(* IEC 61131-3 sources: elnaProjects/kc6/build_BaseProject_ecl/_ (part 5) *)

  (* [A2-14, AI0-1] T_medi_statora_faza_2 *)
  stAI_Ini(data_Ini := TRUE,  dLL := 0.0, dHL := 150.0,
  ISVALIDREF_HW := TRUE, dHW := 130.0, aperturFilter:= 0.5,
  strAI := ai.TStalisStatoraKanal2);
  inits := inits + BOOL_TO_UINT(stAI_Ini.Init);

  (* [A2-14, AI0-2] T_medi_statora_faza_3 *)
  stAI_Ini(data_Ini := TRUE,  dLL := 0.0, dHL :=150.0,
  ISVALIDREF_HW := TRUE, dHW := 130.0, aperturFilter:= 0.5,
  strAI := ai.TStalisStatoraKanal3);
  inits := inits + BOOL_TO_UINT(stAI_Ini.Init);

  (* [A2-14, AI0-3] T_stali_statora_faza_1 *)
  stAI_Ini(data_Ini := TRUE,  dLL := 0.0, dHL := 150.0,
  ISVALIDREF_HW := TRUE, dHW := 130.0, aperturFilter:= 0.5,
  strAI := ai.TMediStatoraKanal1);
  inits := inits + BOOL_TO_UINT(stAI_Ini.Init);

  (********************************************* Модуль A2-15 ******************************************************)

  (* [A2-15, AI1-0] T_stali_statora_faza_2 *)
  stAI_Ini(data_Ini :=TRUE,  dLL := 0.0, dHL := 150.0,
  ISVALIDREF_HW := TRUE, dHW := 130.0, aperturFilter:= 0.5,
  strAI := ai.TMediStatoraKanal2);
  inits := inits + BOOL_TO_UINT(stAI_Ini.Init);

  (* [A2-15, AI1-1] T_stali_statora_faza_3 *)
  stAI_Ini(data_Ini := TRUE,  dLL := 0.0, dHL := 150.0,
  ISVALIDREF_HW := TRUE, dHW := 130.0, aperturFilter:= 0.5,
  strAI := ai.TMediStatoraKanal3);
  inits := inits + BOOL_TO_UINT(stAI_Ini.Init);

  (* [A2-15, AI1-2] T_goryachego_vozdyha_ed_t1 *)
  stAI_Ini(data_Ini := TRUE,  dLL := 0.0, dHL := 100.0,
  ISVALIDREF_HW := TRUE, dHW := 70.0, aperturFilter:= 0.5,
  strAI := ai.TOpornogoPodshipnikaEDT_1);
  inits := inits + BOOL_TO_UINT(stAI_Ini.Init);

  (* [A2-15, AI1-3]  T_goryachego_vozdyha_ed_t2 *)
  stAI_Ini(data_Ini := TRUE,  dLL := 0.0, dHL := 100.0,
  ISVALIDREF_HW := TRUE, dHW := 70.0, aperturFilter:= 0.5,
  strAI := ai.TOpornoYpornogoPodshipnikaEDT_2);
  inits := inits + BOOL_TO_UINT(stAI_Ini.Init);

  (********************************************* Модуль A3-1 ******************************************************)

  (* [A3-1, AI2-0]  T_holodnogo_vozdyha_ed_t1 *)
  stAI_Ini(data_Ini := TRUE,  dLL := 0.0, dHL := 100.0,
  ISVALIDREF_HW := TRUE, dHW := 70.0, aperturFilter:= 0.5,
  strAI := ai.TOpornoYpornogoPodshipnikaKolesaRedEDT_3);
  inits := inits + BOOL_TO_UINT(stAI_Ini.Init);

  (* [A3-1, AI2-1] T_holodnogo_vozdyha_ed_t2 *)
  stAI_Ini(data_Ini := TRUE,  dLL := 0.0, dHL := 100.0,
  ISVALIDREF_HW := TRUE, dHW := 70.0, aperturFilter:= 0.5,
  strAI := ai.TOpornoYpornogoPodshipnikaKolesaRedHT_4);
  inits := inits + BOOL_TO_UINT(stAI_Ini.Init);

  (* [A3-1, AI2-2] T_opornogo_podshipnika_electro_dvigatelia_t1 *)
  stAI_Ini(data_Ini := TRUE,  dLL := 0.0, dHL := 100.0,
  ISVALIDREF_HA := TRUE, ISVALIDREF_HW := TRUE, dHA := 80.0, dHW := 75.0, aperturFilter:= 0.5,
  strAI := ai.TOpornogoPodshipnikaShesterniReduktoraT_5);
  inits := inits + BOOL_TO_UINT(stAI_Ini.Init);

  (* [A3-1, AI2-3] T_opornogo_ypornogo_podshipnika_electro_dvigatelia_so_storony_redyctora_t2 *)
  stAI_Ini(data_Ini := TRUE,  dLL := 0.0, dHL := 100.0,
  ISVALIDREF_HA := TRUE, ISVALIDREF_HW := TRUE, dHA := 80.0, dHW := 75.0, aperturFilter:= 0.5,
  strAI := ai.TOpornogoPodshipnikaReduktoraHT_6);
  inits := inits + BOOL_TO_UINT(stAI_Ini.Init);

  (********************************************* Модуль A3-2 ******************************************************)

  (* [A3-2, AI3-01]  T_oporno_ypornogo_podshipnika_kolesa_redyctora_so_storony_electro_dvigatelya_t3 *)
  stAI_Ini(data_Ini := TRUE,  dLL := 0.0, dHL := 100.0,
  ISVALIDREF_HA := TRUE, ISVALIDREF_HW := TRUE, dHA := 80.0, dHW := 75.0, aperturFilter:= 0.5,
  strAI := ai.TOpornoYpornogoPodshipnikaNagnetateljaT_7_1);
  inits := inits + BOOL_TO_UINT(stAI_Ini.Init);

  (* [A3-2, AI3-1]  T_opornogo_podshipnika_kolesa_redyctora_so_storony_nagnetatelya_t4 *)
  stAI_Ini(data_Ini := TRUE,  dLL := 0.0, dHL := 100.0, aperturFilter:= 0.5,
  ISVALIDREF_HA := TRUE, ISVALIDREF_HW := TRUE, dHA := 80.0, dHW := 75.0,
  strAI := ai.TOpornoYpornogoPodshipnikaNagnetateljaT_7_2);
  inits := inits + BOOL_TO_UINT(stAI_Ini.Init);

  (* [A3-2, AI3-2]  Т подшипника редуктора, т4 *)
  stAI_Ini(data_Ini := TRUE,  dLL := 0.0, dHL := 100.0,
  ISVALIDREF_HA := TRUE, ISVALIDREF_HW := TRUE, dHA := 80.0, dHW := 75.0, aperturFilter:= 0.5,
  strAI := ai.TOpornoYpornogoPodshipnikaSvobodnogoKoncaNT_8_1);
  inits := inits + BOOL_TO_UINT(stAI_Ini.Init);

  (* [A3-2, AI3-3]  Т опорного подшипника нагнетателя, т1 *)
  stAI_Ini(data_Ini := TRUE,  dLL := 0.0, dHL := 100.0,
  ISVALIDREF_HA := TRUE, ISVALIDREF_HW := TRUE, dHA := 80.0, dHW := 75.0, aperturFilter:= 0.5,
  strAI := ai.TOpornoYpornogoPodshipnikaSvobodnogoKoncaNT_8_2);
  inits := inits + BOOL_TO_UINT(stAI_Ini.Init);

  (********************************************* Модуль A3-3 ******************************************************)

  (* [A3-3, AI4-1]  T_oporno_ypornogo_podshipnika_nagnetatelya_so_storony_redyctora_t7_osnovnoi *)
  stAI_Ini(data_Ini := TRUE,  dLL := 0.0, dHL := 100.0,
  ISVALIDREF_HA := TRUE, ISVALIDREF_HW := TRUE, dHA := 80.0, dHW := 75.0, aperturFilter:= 0.5,
  strAI := ai.TYpornogoPodshipnikaRavKolodokHT_9_1);
  inits := inits + BOOL_TO_UINT(stAI_Ini.Init);

  (* [A3-3, AI4-2]  T_oporno_ypornogo_podshipnika_nagnetatelya_so_storony_redyctora_t7_rezervniy *)
  stAI_Ini(data_Ini := TRUE,  dLL := 0.0, dHL := 100.0,
  ISVALIDREF_HA := TRUE, ISVALIDREF_HW := TRUE, dHA := 80.0, dHW := 75.0, aperturFilter:= 0.5,
  strAI := ai.TYpornogoPodshipnikaRavKolodokHT_9_2);
  inits := inits + BOOL_TO_UINT(stAI_Ini.Init);

  (* [A3-3, AI4-3] T_oporno_ypornogo_podshipnika_svobodnogo_konca_nagnetatelya_t8_osnovnoi *)
  stAI_Ini(data_Ini := TRUE,  dLL := 0.0, dHL := 100.0,
  ISVALIDREF_HA := TRUE, ISVALIDREF_HW := TRUE, dHA := 80.0, dHW := 75.0, aperturFilter:= 0.5,
  strAI := ai.TYpornogoPodshipnikaNerabKolodokHT_10_1);
  inits := inits + BOOL_TO_UINT(stAI_Ini.Init);

  (* [A3-3, AI4-4] T_oporno_ypornogo_podshipnika_svobodnogo_konca_nagnetatelya_t8_rezervniy *)
  stAI_Ini(data_Ini := TRUE,  dLL := 0.0, dHL := 100.0,
  ISVALIDREF_HA := TRUE, ISVALIDREF_HW := TRUE, dHA := 80.0, dHW := 75.0, aperturFilter:= 0.5,
  strAI := ai.TYpornogoPodshipnikaNerabKolodokHT_10_2);
  inits := inits + BOOL_TO_UINT(stAI_Ini.Init);

  (********************************************* Модуль A3-4 ******************************************************)

  (* [A3-4, AI5-0] T_ypornogo_podshipnika_rabochih_kolodok_nagnetatelya_t9 *)
  stAI_Ini(data_Ini := TRUE,  dLL := 0.0, dHL := 100.0,
  ISVALIDREF_HA := TRUE, ISVALIDREF_HW := TRUE, dHA := 80.0, dHW := 75.0, aperturFilter:= 0.5,
  strAI := ai.THolodnogoVozduhaEDKanall);
  inits := inits + BOOL_TO_UINT(stAI_Ini.Init);

  (* [A3-4, AI5-1] T_ne_rabochih_kolodok_ypornogo_podshipnika_nagnetatelya_t10 *)
  stAI_Ini(data_Ini := TRUE,  dLL := 0.0, dHL := 100.0,
  ISVALIDREF_HA := TRUE, ISVALIDREF_HW := TRUE, dHA := 80.0, dHW := 75.0, aperturFilter:= 0.5,
  strAI := ai.THolodnogoVozduhaEDKanal2);
  inits := inits + BOOL_TO_UINT(stAI_Ini.Init);

  (* [A3-4, AI5-2]  T_gaz_in_nagnetatelia *)
  stAI_Ini(data_Ini := TRUE,  dLL := -50.0, dHL := 100.0,
  ISVALIDREF_HW := TRUE, dHW := 80.0, aperturFilter:= 0.5,
  strAI := ai.TGorjachegoVozduhaEDKanall);
  inits := inits + BOOL_TO_UINT(stAI_Ini.Init);

  (* [A3-4, AI5-3] T_gaz_out_nagnetatelia *)
  stAI_Ini(data_Ini := TRUE,  dLL := -50.0, dHL := 100.0,
  ISVALIDREF_HA := TRUE, ISVALIDREF_HW := TRUE, dHA := 90.0, dHW := 80.0, aperturFilter:= 0.5,
  strAI := ai.TGorjachegoVozduhaEDKanal2);
  inits := inits + BOOL_TO_UINT(stAI_Ini.Init);

  (********************************************* Модуль A3-5 ******************************************************)

  (* [A3-5, AI6-0] T_masla_do_ABO *)
  stAI_Ini(data_Ini := TRUE,  dLL := 0.0, dHL := 100.0,
  ISVALIDREF_HW := TRUE, dHW := 55.0, aperturFilter:= 0.5,
  strAI := ai.TNArujnogoVozduha);
  inits := inits + BOOL_TO_UINT(stAI_Ini.Init);

  (* [A3-5, AI6-1]  T_masla_posle_ABO *)
  stAI_Ini(data_Ini := TRUE,  dLL := 0.0, dHL := 100.0,
  ISVALIDREF_HW := TRUE, dHW := 55.0, aperturFilter:= 0.5,
  strAI := ai.TgazaNaVhodeH);
  inits := inits + BOOL_TO_UINT(stAI_Ini.Init);

  (* [A3-5, AI6-2] T_masla_v_maslobake *)
  stAI_Ini(data_Ini := TRUE,  dLL := 0.0, dHL := 100.0,
  ISVALIDREF_LW := TRUE, dLW := 25.0, aperturFilter:= 0.5,
  strAI := ai.TgazaNaVyhodeH);
  inits := inits + BOOL_TO_UINT(stAI_Ini.Init);

  (********************************************* Модуль A3-6 ******************************************************)

  (* [A3-6, AI7-0] T_masla_v_maslobake_nad_ten *)
  stAI_Ini(data_Ini := TRUE,  dLL := 0.0, dHL := 100.0,
  ISVALIDREF_HW := TRUE, dHW := 60.0, aperturFilter:= 0.5,
  strAI := ai.T_masla_v_maslobake_nad_ten);
  inits := inits + BOOL_TO_UINT(stAI_Ini.Init);

  (* [A3-6, AI7-1] T_naryjnogo_vozdyxa_rezervniy *)
  stAI_Ini(data_Ini := TRUE,  dLL := -50.0, dHL := 100.0,
  aperturFilter:= 0.5,
  strAI := ai.T_naryjnogo_vozdyxa);
  inits := inits + BOOL_TO_UINT(stAI_Ini.Init);

  (* [A3-6, AI7-2] T_vozduha_V_shkafy *)
  stAI_Ini(data_Ini := TRUE,  dLL := -50.0, dHL := 100.0,
  aperturFilter:= 0.5,
  strAI := ai.T_vozduha_V_shkaf);
  inits := inits + BOOL_TO_UINT(stAI_Ini.Init);

  (********************************************* Модуль A3-8 ******************************************************)

  (* [A3-8, AI9-0]  Davlenie_impylsnogo_gaza *)
  stAI_Ini(data_Ini := TRUE,  dLL := 0.0, dHL := 10.0,
  ISVALIDREF_LW := TRUE, dLW := 5.0, aperturFilter:= 0.5,
  strAI := ai.Davlenie_impylsnogo_gaza);
  inits := inits + BOOL_TO_UINT(stAI_Ini.Init);

  (* [A3-8, AI9-1]  Yroven_masla_v_maslobake *)
  stAI_Ini(data_Ini := TRUE,  dLL := 340.0, dHL := 960.0,
  ISVALIDREF_LW := TRUE, dLW := 350.0, aperturFilter:= 0.5,
  strAI := ai.Yroven_masla_v_maslobake);
  inits := inits + BOOL_TO_UINT(stAI_Ini.Init);

  (* [A3-8, AI9-2]  Osevoi_sdvig_nagnetatelya_vpravo *)
  stAI_Ini(data_Ini := TRUE,  dLL := 0.0, dHL := 1000.0,
  ISVALIDREF_HA := TRUE, ISVALIDREF_HW := TRUE, dHA := 300.0, dHW := 200.0, aperturFilter:= 0.5,
  strAI := ai.Osevoi_sdvig_nagnetatelya_vpravo);
  inits := inits + BOOL_TO_UINT(stAI_Ini.Init);

  (* [A3-8, AI9-3]  Osevoi_sdvig_nagnetatelya_vlevo *)
  stAI_Ini(data_Ini := TRUE,  dLL := 0.0, dHL := 1000.0,
  ISVALIDREF_LA := TRUE, ISVALIDREF_LW := TRUE, dHA := 300.0, dHW := 200.0, aperturFilter:= 0.5,
  strAI := ai.Osevoi_sdvig_nagnetatelya_vlevo);
  inits := inits + BOOL_TO_UINT(stAI_Ini.Init);

  (********************************************* Модуль A3-9 ******************************************************)

  (* [A3-9, AI10-0]  Tok_statora *)
  stAI_Ini(data_Ini := TRUE,  dLL := 0.0, dHL := 1000.0,
  ISVALIDREF_LW := TRUE, dLW := 240.0, aperturFilter:= 0.5,
  strAI := ai.Tok_statora);
  inits := inits + BOOL_TO_UINT(stAI_Ini.Init);

  (* [A3-9, AI10-1]  Kontrol_220_perem *)
  stAI_Ini(data_Ini := TRUE,  dLL := 0.0, dHL := 250.0, aperturFilter:= 0.5,
  ISVALIDREF_LW := TRUE, ISVALIDREF_HW := TRUE,
  dLW := 187.0, dHW := 242.0,
  strAI := ai.Kontrol_220_perem);
  inits := inits + BOOL_TO_UINT(stAI_Ini.Init);

  (* [A3-9, AI10-2] Kontrol_220_post *)
  stAI_Ini(data_Ini := TRUE,  dLL := 0.0, dHL := 250.0, aperturFilter:= 0.5,
  ISVALIDREF_LW := TRUE, ISVALIDREF_HW := TRUE,
  dLW := 187.0, dHW := 242.0,
  strAI := ai.Kontrol_220_post);
  inits := inits + BOOL_TO_UINT(stAI_Ini.Init);

  (********************************************* Модуль A3-10 ******************************************************)

  (* [A3-10, AI11-0] Davlenie_gaza_na_vhode_nagnetatelya *)
  stAI_Ini(data_Ini := TRUE,  dLL := 0.0, dHL := 10.0,
  ISVALIDREF_LW := TRUE, dLW := 5.0, (*ISVALIDREF_LA := TRUE, dLA := 4.6,*) aperturFilter:= 0.5,
  strAI := ai.Davlenie_gaza_na_vhode_nagnetatelya);
  inits := inits + BOOL_TO_UINT(stAI_Ini.Init);

  (* [A3-10, AI11-1] Davlenie_gaza_na_vihode_nagnetatelya *)
  stAI_Ini(data_Ini := TRUE,  dLL := 0.0, dHL := 10.0,
  ISVALIDREF_HW := TRUE, dHW := 7.55, (*ISVALIDREF_HA := TRUE, dHA := 7.65,*) aperturFilter:= 0.5,
  strAI := ai.Davlenie_gaza_na_vihode_nagnetatelya);
  inits := inits + BOOL_TO_UINT(stAI_Ini.Init);

  (* [A3-10, AI11-2] Perepad_davleniya_maslo_gaz *)
  stAI_Ini(data_Ini := TRUE,  dLL := 0.0, dHL := 1600.0,
  ISVALIDREF_LW := TRUE, dLW := 150.0, ISVALIDREF_LA := TRUE, dLA := 100.0,
  strAI := ai.Perepad_davleniya_maslo_gaz);
  inits := inits + BOOL_TO_UINT(stAI_Ini.Init);

  (* [A3-10, AI11-3] Davlenie_masla_posle_nasosa_yplotneniya *)
  stAI_Ini(data_Ini := TRUE,  dLL := 0.0, dHL := 10.0, aperturFilter:= 0.5,
  strAI := ai.Davlenie_masla_posle_nasosa_yplotneniya);
  inits := inits + BOOL_TO_UINT(stAI_Ini.Init);

  (********************************************* Модуль A3-11 ******************************************************)

  (* [A3-11, AI12-0]  Davlenie_masla_smazki_nizkoe *)
  stAI_Ini(data_Ini := TRUE,  dLL := 0.0, dHL := 1000.0,
  ISVALIDREF_LW := TRUE, dLW := 50.0, ISVALIDREF_LA := TRUE, dLA := 25.0,
  strAI := ai.Davlenie_masla_smazki_nizkoe);
  inits := inits + BOOL_TO_UINT(stAI_Ini.Init);

  (* [A3-11, AI12-1]  Davlenie_masla_smazki_visokoe *)
  stAI_Ini(data_Ini := TRUE,  dLL := 0.0, dHL := 1000.0,
  ISVALIDREF_LW := TRUE, dLW := 300.0, ISVALIDREF_LA := TRUE, dLA := 250.0,
  strAI := ai.Davlenie_masla_smazki_visokoe);
  inits := inits + BOOL_TO_UINT(stAI_Ini.Init);

  (* [A3-11, AI12-2]  Davlenie_masla_smazki_posle_GNS *)
  stAI_Ini(data_Ini := TRUE,  dLL := 0.0, dHL := 1000.0,
  ISVALIDREF_LW := TRUE, dLW := 400.0, aperturFilter:= 0.5,
  strAI := ai.Davlenie_masla_smazki_posle_GNS);
  inits := inits + BOOL_TO_UINT(stAI_Ini.Init);

  (* [A3-11, AI12-3]  Perepad_davleniya_gaza_na_konfyzore *)
  stAI_Ini(data_Ini := TRUE,  dLL := 0.0, dHL := 250.0, aperturFilter:= 0.5,
  strAI := ai.Perepad_davleniya_gaza_na_konfyzore);
  inits := inits + BOOL_TO_UINT(stAI_Ini.Init);

  (********************************************* Модуль A3-12 ******************************************************)

  (* [A3-12, AI13-0] Perepad_davleniya_masla_na_maslyanom_filtre *)
  stAI_Ini(data_Ini := TRUE,  dLL := 0.0, dHL := 250.0,
  ISVALIDREF_HW := TRUE, dHW := 150.0, aperturFilter:= 0.5,
  strAI := ai.Perepad_davleniya_masla_na_maslyanom_filtre);
  inits := inits + BOOL_TO_UINT(stAI_Ini.Init);

  (********************************************* Модуль A3-13 ******************************************************)

  (* [A3-13, AI14-0]  Vibroploskost_opornogo_podshipnika_electro_dvigatelya_t1 *)
  stAI_Ini(data_Ini := TRUE,  dLL := 0.0, dHL := 25.0,
  ISVALIDREF_HW := TRUE, ISVALIDREF_HA := TRUE, dHW := 11.0, dHA := 18.0,
  strAI := ai.Vibroskorost_OP_ED_t1);
  inits := inits + BOOL_TO_UINT(stAI_Ini.Init);

  (* [A3-13, AI14-1]  Vibroploskost_oporno_ypornogo_podshipnika_electro_dvigatelya_so_storony_redyctora_t2 *)
  stAI_Ini(data_Ini := TRUE,  dLL := 0.0, dHL := 25.0,
  ISVALIDREF_HW := TRUE, ISVALIDREF_HA := TRUE, dHW := 11.0, dHA := 18.0, aperturFilter:= 0.5,
  strAI := ai.Vibroskorost_OYP_ED_so_storony_redyctora_t2);
  inits := inits + BOOL_TO_UINT(stAI_Ini.Init);

  (* [A3-13, AI14-2]  Vibroploskost_oporno_ypornogo_podshipnika_kolesa_redyktora_so_storony_electro_dvigatelya_t3 *)
  stAI_Ini(data_Ini := TRUE,  dLL := 0.0, dHL := 25.0,
  ISVALIDREF_HW := TRUE, ISVALIDREF_HA := TRUE, dHW := 11.0, dHA := 18.0, aperturFilter:= 0.5,
  strAI := ai.Vibroskorost_OYP_kolesa_ED_t3);
  inits := inits + BOOL_TO_UINT(stAI_Ini.Init);

  (* [A3-13, AI14-3]  Vibroploskost_oporno_ypornogo_podshipnika_kolesa_redyktora_so_storony_nagnetatelya_t4_rezerv *)
  stAI_Ini(data_Ini := TRUE,  dLL := 0.0, dHL := 25.0,
  ISVALIDREF_HW := TRUE, ISVALIDREF_HA := TRUE, dHW := 11.0, dHA := 18.0, aperturFilter:= 0.5,
  strAI := ai.Vibroskorost_OP_kolesa_nagnetatelya_t4);
  inits := inits + BOOL_TO_UINT(stAI_Ini.Init);

  (********************************************* Модуль A3-14 ******************************************************)

  (* [A3-14, AI15-0]  Vibroploskost_opornogo_podshipnika_shesterni_redyktora_so_storony_nagnetatelya_t5_rezerv *)
  stAI_Ini(data_Ini := TRUE,  dLL := 0.0, dHL := 25.0,
  ISVALIDREF_HW := TRUE, ISVALIDREF_HA := TRUE, dHW := 11.0, dHA := 18.0, aperturFilter:= 0.5,
  strAI := ai.Vibroskorost_OP_shesterni_ED_t5);
  inits := inits + BOOL_TO_UINT(stAI_Ini.Init);

  (* [A3-14, AI15-1]  Vibroploskost_opornogo_podshipnika_shesterni_redyktora_so_storony_nagnetatelya_t6 *)
  stAI_Ini(data_Ini := TRUE,  dLL := 0.0, dHL := 25.0,
  ISVALIDREF_HW := TRUE, ISVALIDREF_HA := TRUE, dHW := 11.0, dHA := 18.0, aperturFilter:= 0.5,
  strAI := ai.Vibroskorost_OP_shesterni_nagnetatelya_t6);
  inits := inits + BOOL_TO_UINT(stAI_Ini.Init);

  initiales := 0;
  IF init THEN initiales := inits; END_IF;
END_FUNCTION_BLOCK

FUNCTION_BLOCK proc_AO
  VAR
    fb_Reserv_AO_1 : fb_AOSourceMlp;
    fb_Reserv_AO_2 : fb_AOSourceMlp;
  END_VAR
  VAR_EXTERNAL
    ao : AOConfig;
    arAOUT_0 : TDoubleData;
    arAOUT_1 : TDoubleData;
  END_VAR

  (* Циклический опрос. Входные аналоговые параметры *)

  (* Модуль A10 *)

  (* [A10-1, AO0] Резерв (A10) *)
  fb_Reserv_AO_1(OutCurrent := arAOUT_0, strAO := ao.Reserv_AO_1);

  (* [A10-1, AO1] Резерв (A10) *)
  fb_Reserv_AO_2(OutCurrent := arAOUT_1, strAO := ao.Reserv_AO_2);
END_FUNCTION_BLOCK

FUNCTION_BLOCK proc_AO_Init
  VAR_INPUT
    init : BOOL;
  END_VAR
  VAR
    stAO_Ini : fb_AO_Init;
    inits : UINT;
  END_VAR
  VAR_INPUT
    initiales : UINT;
  END_VAR
  VAR_EXTERNAL
    ao : AOConfig;
  END_VAR

  (* Инициализация начало. Входные аналоговые параметры *)

  inits := 0; (* Флаг необходимости инициализации структур-дескрипторов *)

  (* Модуль A10 *)
  (* [A10, AO0] Резерв (A) *)
  stAO_Ini(data_Ini := TRUE, (*outLL := 4000.0, outHL := 20000.0,*)
    newLL_ISVALIDREF := TRUE, newHL_ISVALIDREF := TRUE,
    newLL := 0.0, newHL := 100.0,
    strAO := ao.Reserv_AO_1);
  inits := inits + BOOL_TO_UINT(stAO_Ini.Init);

  (* [A1-10, AO1] Резерв (A) *)
  stAO_Ini(data_Ini := TRUE, (*outLL := 4000.0, outHL := 20000.0,*)
    (*newLL_ISVALIDREF := TRUE, newHL_ISVALIDREF := TRUE,*)
    (*newLL := 0.0, newHL := 100.0,*)
  strAO := ao.Reserv_AO_2);
  inits := inits + BOOL_TO_UINT(stAO_Ini.Init);

  initiales := 0;
  IF init THEN initiales := inits; END_IF;
END_FUNCTION_BLOCK

FUNCTION_BLOCK proc_DI
  VAR_EXTERNAL
    di : DiConfig;
  END_VAR
  VAR
    di_0 : fb_DiSourceMlp;
    di_1 : fb_DiSourceMlp;
    di_2 : fb_DiSourceMlp;
    di_3 : fb_DiSourceMlp;
    di_4 : fb_DiSourceMlp;
    di_5 : fb_DiSourceMlp;
    di_6 : fb_DiSourceMlp;
    di_7 : fb_DiSourceMlp;
    di_8 : fb_DiSourceMlp;
    di_9 : fb_DiSourceMlp;
    di_10 : fb_DiSourceMlp;
    di_11 : fb_DiSourceMlp;
    di_12 : fb_DiSourceMlp;
    di_13 : fb_DiSourceMlp;
    di_14 : fb_DiSourceMlp;
    di_15 : fb_DiSourceMlp;
    di_16 : fb_DiSourceMlp;
    di_17 : fb_DiSourceMlp;
  END_VAR
  VAR_EXTERNAL
    arDIN_0 : TItemDIN;
    arDIN_1 : TItemDIN;
    arDIN_2 : TItemDIN;
    arDIN_3 : TItemDIN;
    arDIN_4 : TItemDIN;
    arDIN_5 : TItemDIN;
    arDIN_6 : TItemDIN;
    arDIN_7 : TItemDIN;
    arDIN_8 : TItemDIN;
    arDIN_9 : TItemDIN;
    arDIN_10 : TItemDIN;
    arDIN_11 : TItemDIN;
    arDIN_12 : TItemDIN;
    arDIN_13 : TItemDIN;
    arDIN_14 : TItemDIN;
    arDIN_15 : TItemDIN;
    arDIN_16 : TItemDIN;
    arDIN_17 : TItemDIN;
    arERR_1 : TItemDIN;
    arERR_2 : TItemDIN;
    arERR_3 : TItemDIN;
    arERR_4 : TItemDIN;
    arERR_5 : TItemDIN;
    arERR_6 : TItemDIN;
    arERR_7 : TItemDIN;
    arERR_8 : TItemDIN;
    arERR_0 : TItemDIN;
    arERR_9 : TItemDIN;
    arERR_10 : TItemDIN;
    arERR_11 : TItemDIN;
    arERR_12 : TItemDIN;
    arERR_13 : TItemDIN;
    arERR_14 : TItemDIN;
    arERR_15 : TItemDIN;
    arERR_16 : TItemDIN;
    arERR_17 : TItemDIN;
    DI_A1_10_wValue : UINT;
    DI_A1_11_wValue : UINT;
    DI_A1_12_wValue : UINT;
    DI_A1_13_wValue : UINT;
    DI_A1_14_wValue : UINT;
    DI_A1_15_wValue : UINT;
    DI_A1_1_wValue : UINT;
    DI_A1_2_wValue : UINT;
    DI_A1_3_wValue : UINT;
    DI_A1_4_wValue : UINT;
    DI_A1_5_wValue : UINT;
    DI_A1_6_wValue : UINT;
    DI_A1_7_wValue : UINT;
    DI_A1_8_wValue : UINT;
    DI_A1_9_wValue : UINT;
    DI_A2_1_wValue : UINT;
    DI_A2_2_wValue : UINT;
    DI_A2_3_wValue : UINT;
    A1_10_err_mode : UINT;
    A1_11_err_mode : UINT;
    A1_12_err_mode : UINT;
    A1_13_err_mode : UINT;
    A1_14_err_mode : UINT;
    A1_15_err_mode : UINT;
    A1_1_err_mode : UINT;
    A1_2_err_mode : UINT;
    A1_3_err_mode : UINT;
    A1_4_err_mode : UINT;
    A1_5_err_mode : UINT;
    A1_6_err_mode : UINT;
    A1_7_err_mode : UINT;
    A1_8_err_mode : UINT;
    A1_9_err_mode : UINT;
    A2_1_err_mode : UINT;
    A2_2_err_mode : UINT;
    A2_3_err_mode : UINT;
  END_VAR

  (* Циклический опрос. Входные дискретные параметры *)

  (* Модуль A1-1 *)
  di_0(arDIN := arDIN_0, strDI:=di.di_0, err_mod:=arERR_0);
  DI_A1_1_wValue:=arDIN_0.wValue;
  A1_1_err_mode :=arERR_0.wValue;

  (* Модуль A1-2 *)
  di_1(arDIN := arDIN_1, strDI:=di.di_1, err_mod:=arERR_1);
  DI_A1_2_wValue:=arDIN_1.wValue;
  A1_2_err_mode :=arERR_1.wValue;

  (* Модуль A1-3 *)
  di_2(arDIN := arDIN_2, strDI:=di.di_2,  err_mod:=arERR_2);
  DI_A1_3_wValue:=arDIN_2.wValue;
  A1_3_err_mode :=arERR_2.wValue;

  (* Модуль A1-4 *)
  di_3(arDIN := arDIN_3, strDI:=di.di_3,  err_mod:=arERR_3);
  DI_A1_4_wValue:=arDIN_3.wValue;
  A1_4_err_mode :=arERR_3.wValue;

  (* Модуль A1-5 *)
  di_4(arDIN := arDIN_4, strDI:=di.di_4,  err_mod:=arERR_4);
  DI_A1_5_wValue:=arDIN_4.wValue;
  A1_5_err_mode :=arERR_4.wValue;

  (* Модуль A1-6 *)
  di_5(arDIN := arDIN_5, strDI:=di.di_5,  err_mod:=arERR_5);
  DI_A1_6_wValue:=arDIN_5.wValue;
  A1_6_err_mode :=arERR_5.wValue;

  (* Модуль A1-7 *)
  di_6(arDIN := arDIN_6, strDI:=di.di_6,  err_mod:=arERR_6);
  DI_A1_7_wValue:=arDIN_6.wValue;
  A1_7_err_mode :=arERR_6.wValue;

  (* Модуль A1-8 *)
  di_7(arDIN := arDIN_7, strDI:=di.di_7,  err_mod:=arERR_7);
  DI_A1_8_wValue:=arDIN_7.wValue;
  A1_8_err_mode :=arERR_7.wValue;

  (* Модуль A1-9 *)
  di_8(arDIN := arDIN_8, strDI:=di.di_8,  err_mod:=arERR_8);
  DI_A1_9_wValue:=arDIN_8.wValue;
  A1_9_err_mode :=arERR_8.wValue;

  (* Модуль A1-10 *)
  di_9(arDIN := arDIN_9, strDI:=di.di_9,  err_mod:=arERR_9);
  DI_A1_10_wValue:=arDIN_9.wValue;
  A1_10_err_mode :=arERR_9.wValue;

  (* Модуль A1-11 *)
  di_10(arDIN := arDIN_10, strDI:=di.di_10,  err_mod:=arERR_10);
  DI_A1_11_wValue:=arDIN_10.wValue;
  A1_11_err_mode :=arERR_10.wValue;

  (* Модуль A1-12 *)
  di_11(arDIN := arDIN_11, strDI:=di.di_11,  err_mod:=arERR_11);
  DI_A1_12_wValue:=arDIN_11.wValue;
  A1_12_err_mode :=arERR_11.wValue;

  (* Модуль A1-13 *)
  di_12(arDIN := arDIN_12, strDI:=di.di_12,  err_mod:=arERR_12);
  DI_A1_13_wValue:=arDIN_12.wValue;
  A1_13_err_mode :=arERR_12.wValue;

  (* Модуль A1-14 *)
  di_13(arDIN := arDIN_13, strDI:=di.di_13,  err_mod:=arERR_13);
  DI_A1_14_wValue:=arDIN_13.wValue;
  A1_14_err_mode :=arERR_13.wValue;

  (* Модуль A1-15 *)
  di_14(arDIN := arDIN_14, strDI:=di.di_14,  err_mod:=arERR_14);
  DI_A1_15_wValue:=arDIN_14.wValue;
  A1_15_err_mode :=arERR_14.wValue;

  (* Модуль A2-1 *)
  di_15(arDIN := arDIN_15, strDI:=di.di_15,  err_mod:=arERR_15);
  DI_A2_1_wValue:=arDIN_15.wValue;
  A2_1_err_mode :=arERR_15.wValue;

  (* Модуль A2-2 *)
  di_16(arDIN := arDIN_16, strDI:=di.di_16,  err_mod:=arERR_16);
  DI_A2_2_wValue:=arDIN_16.wValue;
  A2_2_err_mode :=arERR_16.wValue;

  (* Модуль A2-3 *)
  di_17(arDIN := arDIN_17, strDI:=di.di_17,  err_mod:=arERR_17);
  DI_A2_3_wValue:=arDIN_17.wValue;
  A2_3_err_mode :=arERR_17.wValue;
END_FUNCTION_BLOCK

FUNCTION_BLOCK proc_DI_Init
  VAR_INPUT
    init : BOOL;
  END_VAR
  VAR
    stDI_Ini : fb_DI_Init;
    inits : UINT;
  END_VAR
  VAR_INPUT
    initiales : UINT;
  END_VAR
  VAR_EXTERNAL
    di : DiConfig;
  END_VAR

  (* Инициализация начало. Входные дискретные параметры *)

  inits := 0; (* Флаг необходимости инициализации структур-дескрипторов *)

  (* Модуль A1-1 *)

  stDI_Ini(data_Ini := true, imit:=FALSE, strDI := di.di_0);
  inits := inits + BOOL_TO_UINT(stDI_Ini.Init);

  stDI_Ini(data_Ini := true, imit:=FALSE, strDI := di.di_1);
  inits := inits + BOOL_TO_UINT(stDI_Ini.Init);

  (* Модуль A1-2 *)
  stDI_Ini(data_Ini := true, imit:=FALSE, strDI := di.di_2);
  inits := inits + BOOL_TO_UINT(stDI_Ini.Init);

  stDI_Ini(data_Ini := true, imit:=FALSE, strDI := di.di_3);
  inits := inits + BOOL_TO_UINT(stDI_Ini.Init);

  (* Модуль A1-3 *)
  stDI_Ini(data_Ini := true, imit:=FALSE, strDI := di.di_4);
  inits := inits + BOOL_TO_UINT(stDI_Ini.Init);

  stDI_Ini(data_Ini := true, imit:=FALSE, strDI := di.di_5);
  inits := inits + BOOL_TO_UINT(stDI_Ini.Init);

  (* Модуль A1-4 *)
  stDI_Ini(data_Ini := true, imit:=FALSE, strDI := di.di_6);
  inits := inits + BOOL_TO_UINT(stDI_Ini.Init);

  stDI_Ini(data_Ini := true, imit:=FALSE, strDI := di.di_7);
  inits := inits + BOOL_TO_UINT(stDI_Ini.Init);

  (* Модуль A1-5 *)
  stDI_Ini(data_Ini := true, imit:=FALSE,  strDI := di.di_8);
  inits := inits + BOOL_TO_UINT(stDI_Ini.Init);

  stDI_Ini(data_Ini := true, imit:=FALSE,  strDI := di.di_9);
  inits := inits + BOOL_TO_UINT(stDI_Ini.Init);

  (* Модуль A1-6 *)
  stDI_Ini(data_Ini := true, imit:=FALSE,  strDI := di.di_10);
  inits := inits + BOOL_TO_UINT(stDI_Ini.Init);

  stDI_Ini(data_Ini := true, imit:=FALSE,  strDI := di.di_11);
  inits := inits + BOOL_TO_UINT(stDI_Ini.Init);

  (* Модуль A1-7 *)
  stDI_Ini(data_Ini := true, imit:=FALSE, strDI := di.di_12);
  inits := inits + BOOL_TO_UINT(stDI_Ini.Init);

  stDI_Ini(data_Ini := true, imit:=FALSE, strDI := di.di_13);
  inits := inits + BOOL_TO_UINT(stDI_Ini.Init);

  (* Модуль A1-8 *)
  stDI_Ini(data_Ini := true, imit:=FALSE, strDI := di.di_14);
  inits := inits + BOOL_TO_UINT(stDI_Ini.Init);

  stDI_Ini(data_Ini := true, imit:=FALSE, strDI := di.di_15);
  inits := inits + BOOL_TO_UINT(stDI_Ini.Init);

  initiales := 0;
  IF init THEN initiales := inits; END_IF;
END_FUNCTION_BLOCK

FUNCTION_BLOCK proc_DO
  VAR_EXTERNAL
    od : DOconfig;
  END_VAR
  VAR
    do_0 : fb_DOSourceMlp;
    do_1 : fb_DOSourceMlp;
    do_2 : fb_DOSourceMlp;
    do_3 : fb_DOSourceMlp;
    do_4 : fb_DOSourceMlp;
    do_5 : fb_DOSourceMlp;
    do_6 : fb_DOSourceMlp;
    do_7 : fb_DOSourceMlp;
    do_8 : fb_DOSourceMlp;
    do_9 : fb_DOSourceMlp;
    gpio_out : fb_DOSourceMlp;
  END_VAR
  VAR_EXTERNAL
    arERR_18 : TItemDIN;
    arERR_19 : TItemDIN;
    arERR_20 : TItemDIN;
    arERR_21 : TItemDIN;
    arERR_22 : TItemDIN;
    arERR_23 : TItemDIN;
    arERR_24 : TItemDIN;
    arERR_25 : TItemDIN;
    arERR_26 : TItemDIN;
    arERR_27 : TItemDIN;
    arDOUT_0 : TWordData;
    arDOUT_1 : TWordData;
    arDOUT_2 : TWordData;
    arDOUT_3 : TWordData;
    arDOUT_4 : TWordData;
    arDOUT_5 : TWordData;
    arDOUT_6 : TWordData;
    arDOUT_7 : TWordData;
    arDOUT_8 : TWordData;
    arDOUT_9 : TWordData;
    arERR_66 : TItemDIN;
    arDOUT_66 : TWordData;
    A2_10_err_mode : UINT;
    A2_11_err_mode : UINT;
    A2_12_err_mode : UINT;
    A2_13_err_mode : UINT;
    A2_4_err_mode : UINT;
    A2_5_err_mode : UINT;
    A2_6_err_mode : UINT;
    A2_7_err_mode : UINT;
    A2_8_err_mode : UINT;
    A2_9_err_mode : UINT;
    DO_A2_10_wValue : UINT;
    DO_A2_11_wValue : UINT;
    DO_A2_12_wValue : UINT;
    DO_A2_13_wValue : UINT;
    DO_A2_4_wValue : UINT;
    DO_A2_5_wValue : UINT;
    DO_A2_6_wValue : UINT;
    DO_A2_7_wValue : UINT;
    DO_A2_8_wValue : UINT;
    DO_A2_9_wValue : UINT;
  END_VAR

  (* Циклический опрос. Входные дискретные параметры *)

  (* Модуль A2-4 *)
  do_0(arDout := arDOUT_0, strDO := od.do_0, err_mod:=arERR_18);
  DO_A2_4_wValue:=arDOUT_0.wValue;
  A2_4_err_mode :=arERR_18.wValue;

  (* Модуль A2-5 *)
  do_1(arDout := arDOUT_1, strDO := od.do_1, err_mod:=arERR_19);
  DO_A2_5_wValue:=arDOUT_1.wValue;
  A2_5_err_mode :=arERR_19.wValue;

  (* Модуль A2-6 *)
  do_2(arDout := arDOUT_2, strDO := od.do_2, err_mod:=arERR_20);
  DO_A2_6_wValue:=arDOUT_2.wValue;
  A2_6_err_mode :=arERR_20.wValue;

  (* Модуль A2-7 *)
  do_3(arDout := arDOUT_3, strDO := od.do_3, err_mod:=arERR_21);
  DO_A2_7_wValue:=arDOUT_3.wValue;
  A2_7_err_mode :=arERR_21.wValue;

  (* Модуль A2-8 *)
  do_4(arDout := arDOUT_4, strDO := od.do_4, err_mod:=arERR_22);
  DO_A2_8_wValue:=arDOUT_4.wValue;
  A2_8_err_mode :=arERR_22.wValue;

  (* Модуль A2-9 *)
  do_5(arDout := arDOUT_5, strDO := od.do_5, err_mod:=arERR_23);
  DO_A2_9_wValue:=arDOUT_5.wValue;
  A2_9_err_mode :=arERR_23.wValue;

  (* Модуль A2-10 *)
  do_6(arDout := arDOUT_6, strDO := od.do_6, err_mod:=arERR_24);
  DO_A2_10_wValue:=arDOUT_6.wValue;
  A2_10_err_mode :=arERR_24.wValue;

  (* Модуль A2-11 *)
  do_7(arDout := arDOUT_7, strDO := od.do_7, err_mod:=arERR_25);
  DO_A2_11_wValue:=arDOUT_7.wValue;
  A2_11_err_mode :=arERR_25.wValue;

  (* Модуль A2-12 *)
  do_8(arDout := arDOUT_8, strDO := od.do_8, err_mod:=arERR_26);
  DO_A2_12_wValue:=arDOUT_8.wValue;
  A2_12_err_mode :=arERR_26.wValue;

  (* Модуль A2-13 *)
  do_9(arDout := arDOUT_9, strDO := od.do_9, err_mod:=arERR_27);
  DO_A2_13_wValue:=arDOUT_9.wValue;
  A2_13_err_mode :=arERR_27.wValue;

  gpio_out(arDout := arDOUT_66, strDO := od.gpio_out, err_mod:=arERR_66);
END_FUNCTION_BLOCK

FUNCTION_BLOCK proc_DO_Init
  VAR_INPUT
    init : BOOL;
  END_VAR
  VAR
    stDO_Ini : fb_DO_Init;
    inits : UINT;
  END_VAR
  VAR_INPUT
    initiales : UINT;
  END_VAR
  VAR_EXTERNAL
    od : DOconfig;
  END_VAR

  (* Инициализация начало. Входные дискретные параметры *)

  inits := 0; (* Флаг необходимости инициализации структур-дескрипторов *)

  (* Модуль A1-15 *)
  stDO_Ini(data_Ini := true, imit:=FALSE, strDO := od.do_0);
  inits := inits + BOOL_TO_UINT(stDO_Ini.Init);

  (* Модуль A1-16 *)
  stDO_Ini(data_Ini := true, imit:=FALSE, strDO := od.do_1);
  inits := inits + BOOL_TO_UINT(stDO_Ini.Init);

  (* Модуль A1-17 *)
  stDO_Ini(data_Ini := true, imit:=FALSE, strDO := od.do_2);
  inits := inits + BOOL_TO_UINT(stDO_Ini.Init);

  (* Модуль A1-18 *)
  stDO_Ini(data_Ini := true, imit:=FALSE, strDO := od.do_3);
  inits := inits + BOOL_TO_UINT(stDO_Ini.Init);

  (* Модуль A1-19 *)
  stDO_Ini(data_Ini := true, imit:=FALSE, strDO := od.do_4);
  inits := inits + BOOL_TO_UINT(stDO_Ini.Init);

  (* Модуль A1-20 *)
  stDO_Ini(data_Ini := true, imit:=FALSE, strDO := od.do_5);
  inits := inits + BOOL_TO_UINT(stDO_Ini.Init);

  (* Модуль A1-21 *)
  stDO_Ini(data_Ini := true, imit:=FALSE, strDO := od.do_6);
  inits := inits + BOOL_TO_UINT(stDO_Ini.Init);

  (* Модуль A1-22 *)
  stDO_Ini(data_Ini := true, imit:=FALSE, strDO := od.do_7);
  inits := inits + BOOL_TO_UINT(stDO_Ini.Init);

  (* Модуль A1-23 *)
  stDO_Ini(data_Ini := true, imit:=FALSE, strDO := od.gpio_out);
  inits := inits + BOOL_TO_UINT(stDO_Ini.Init);
  initiales := 0;

  IF init THEN initiales := inits; END_IF;
END_FUNCTION_BLOCK

FUNCTION_BLOCK fb_OilPump
  VAR_INPUT
    statOn : BOOL;
    statOff : BOOL;
    statOn_reliability : BOOL;
    statOff_reliability : BOOL;
  END_VAR
  VAR_IN_OUT
    StrSw : struct_OilPump;
  END_VAR
  VAR_INPUT
    inNs : TYPE_ReliableBit;
    inAccident : TYPE_ReliableBit;
    inLocal : TYPE_ReliableBit;
    inAuto : TYPE_ReliableBit;
    inDistance : TYPE_ReliableBit;
    inBreakCmdOn : TYPE_ReliableBit;
    inBreakCmdOff : TYPE_ReliableBit;
  END_VAR
  VAR
    onInit : BOOL         := FALSE;
    _statOn : BOOL;
    _statOff : BOOL;
    lastOnStatus : BYTE;
    cmd : BYTE;
    source : BYTE;
    lastCmd : BYTE;
    source_for_Status : BYTE;
    cmd_for_Status : BYTE;
    command_error_for_Status : BYTE;
    _sunpackerCommand : fb_sunpackerCommand;
    _statusDualInput : TYPE_statusDualInput;
    _commandDualInput : TYPE_commandDualInput;
    _commandErrorTimer : BOOL;
    resetErrorTimer : BOOL;
    _changWithoutCommand : BOOL;
    errorCMDTimer : TON;
    _errorReset : TON;
    outputsSets : TOF;
  END_VAR
  VAR_IN_OUT
    cmdOn : BOOL;
    cmdOff : BOOL;
  END_VAR

  IF NOT onInit THEN
  IF StrSw.ISVALIDREF_cmdOn XOR StrSw.ISVALIDREF_cmdOff THEN
  	IF 	StrSw.ISVALIDREF_cmdOn THEN
  		lastCmd:= 2; (*baseCmdOff*)
  	ELSE
  		lastCmd:= 1; (*baseCmdOn*)
  	END_IF;
  END_IF;
  onInit:=TRUE;
  END_IF;

  (* ---- Если управление с ВУ заблокировано, то в ИМ передаем команду из алгоритма ---- *)
  IF StrSw.inOpcCommandsDisabled THEN
  	StrSw.inCommand := StrSw.inCommand_Alg;
  ELSE (* иначе передаем команду с АРМа*)
  	StrSw.inCommand := StrSw.inCommand_ARM;
  END_IF;

  (* ---- Формирование состояния механизма ---- *)

  IF (StrSw.ISVALIDREF_statOn) OR (StrSw.ISVALIDREF_statOff) THEN
  	IF (StrSw.ISVALIDREF_statOn) AND (StrSw.ISVALIDREF_statOff) THEN
  	StrSw.reliability:= statOn_reliability AND statOff_reliability;
  		_statOn  := statOn;
  		_statOff := statOff;
  	ELSIF (StrSw.ISVALIDREF_statOn) THEN
                       StrSw.reliability:= statOn_reliability;
  		_statOn  := statOn;
  		_statOff := NOT statOn;
  	ELSIF (StrSw.ISVALIDREF_statOff) THEN
  		 StrSw.reliability:= statOff_reliability;
  		_statOn  := NOT statOff;
  		_statOff :=statOff;
  	END_IF;

  	IF StrSw.reliability THEN
  		IF _statOn AND NOT _statOff 		THEN 	StrSw.onStatus := _statusDualInput.STATUS_ON;
  		ELSIF _statOff AND NOT _statOn 	THEN 	StrSw.onStatus := _statusDualInput.Status_OFF;
  		ELSIF NOT _statOn AND NOT _statOff 	THEN 	StrSw.onStatus := _statusDualInput.STATUS_TRANSITIONAL;
  		ELSE					StrSw.onStatus := _statusDualInput.STATUS_ERROR;
                      END_IF;

  	ELSE
  		StrSw.onStatus := _statusDualInput.STATUS_NOTDEFINED;

  	END_IF;
  ELSE
  	CASE BYTE_TO_INT(lastCmd) OF
  		(*baseCmdOn*) 1: StrSw.onStatus  := _statusDualInput.STATUS_ON;
  		(*baseCmdOff*) 2: StrSw.onStatus  := _statusDualInput.STATUS_OFF;

  	ELSE
  		 StrSw.onStatus := _statusDualInput.STATUS_NOTDEFINED;

  	END_CASE;
  END_IF;

  StrSw.Accident := inAccident.value AND inAccident.reliability;
  StrSw.Ns := inNs.value AND inNs.reliability;
  StrSw.Local := inLocal.value AND inLocal.reliability;
  StrSw.Auto := inAuto.value AND inAuto.reliability;
  StrSw.Distance := inDistance.value AND inDistance.reliability;
  StrSw.OpcCommandsDisabled := StrSw.inOpcCommandsDisabled;

  StrSw.Blocked:=StrSw.Accident OR StrSw.Local OR StrSw.breakCmdOn OR StrSw.breakCmdOff OR StrSw.inBlocked;

  StrSw.Rezervny:=NOT StrSw.Osnovnoy;

  (* ---- Формирование признака сдвига ---- *)
  StrSw.sdvig  := FALSE;
  IF (StrSw.ISVALIDREF_cmdOn OR StrSw.ISVALIDREF_cmdOff) AND NOT StrSw.Local THEN
  	IF cmd = 0 THEN
  		IF (lastOnStatus <> StrSw.onStatus AND
  		(StrSw.onStatus <> _statusDualInput.STATUS_NOTDEFINED AND StrSw.onStatus <> _statusDualInput.STATUS_ERROR) AND
  		(lastOnStatus <> _statusDualInput.STATUS_NOTDEFINED AND lastOnStatus <> _statusDualInput.STATUS_ERROR)) THEN
  			StrSw.sdvig   := TRUE;
  		END_IF;
  	END_IF;
  END_IF;
  lastOnStatus := StrSw.onStatus;

  (* ---- Распаковка команды ---- *)
  _sunpackerCommand(command := StrSw.inCommand);
  	cmd := _sunpackerCommand.cmd;
  	source := _sunpackerCommand.source;

  (* ---- Обработка команды ---- *)
  IF cmd <> 0 AND lastCmd <> cmd and (((NOT StrSw.opcCommandsDisabled) AND source > 0) OR source = 0) then
  	CASE BYTE_TO_INT(cmd) OF
  	(*cmd_open*) 1 :
  			IF  StrSw.ISVALIDREF_cmdOn THEN StrSw.CmdOn := TRUE;
  				IF StrSw.ISVALIDREF_cmdOff THEN StrSw.CmdOff := FALSE; END_IF;
  			ELSIF  StrSw.ISVALIDREF_cmdOff THEN StrSw.CmdOff := FALSE;  END_IF;
  			errorCMDTimer(IN := false);
  			_commandErrorTimer := true;
  			StrSw.lastCmdIsOn := true;
  	(*cmd_close*) 2 :
  			IF StrSw.ISVALIDREF_cmdOff THEN StrSw.CmdOff := TRUE;
  				IF StrSw.ISVALIDREF_cmdOn THEN StrSw.CmdOn := FALSE; END_IF;
  			ELSIF StrSw.ISVALIDREF_cmdOn THEN StrSw.CmdOn := FALSE; END_IF;
  			errorCMDTimer(IN := false);

  			_commandErrorTimer := true;
  			StrSw.lastCmdIsOn := false;
  	(*cmd_reset*) 3 :    IF StrSw.ISVALIDREF_statOn OR StrSw.ISVALIDREF_statOff THEN
  			StrSw.CmdOn := FALSE;
  			StrSw.CmdOff := FALSE;
                                lastCmd := 0;
  			_commandErrorTimer := false;
  			StrSw.lastCmdIsOn := false;
                                 END_IF;
  	END_CASE;
  	source_for_Status := source;
  	cmd_for_Status := cmd;
  	command_error_for_Status := 0;
  END_IF;

  lastCmd := cmd;
  errorCMDTimer(In := _commandErrorTimer, PT :=T#10s);

  (* ---- алгоритм  для команды ВКЛючить ---- *)
  IF (StrSw.onStatus = _statusDualInput.STATUS_ON) and StrSw.lastCmdIsOn then
  	IF StrSw.ISVALIDREF_cmdOn AND StrSw.ISVALIDREF_cmdOff then  StrSw.cmdOn := false; END_IF;

  	 errorCMDTimer(In := false);
  	 _commandErrorTimer := false;
  	 cmd_for_Status := 0;
  	 source_for_Status := 0;
  END_IF;

  (* ---- off ---- *)
  IF (StrSw.onStatus = _statusDualInput.STATUS_OFF) and (NOT StrSw.lastCmdIsOn) then
  	IF StrSw.ISVALIDREF_cmdOn AND StrSw.ISVALIDREF_cmdOff then  StrSw.cmdOff := false; END_IF;

  	 errorCMDTimer(In := false);
  	 _commandErrorTimer := false;
  	 cmd_for_Status := 0;
  	 source_for_Status := 0;
  END_IF;

  (* ---- ошибка исполнения команды ---- *)
  if errorCMDTimer.Q and (cmd_for_Status <> 0) then
  	command_error_for_Status :=  cmd_for_Status;
  	_commandErrorTimer := false;
  	StrSw.CmdOn := false;
  	StrSw.CmdOff := false;
  	lastCmd := 0;
  end_if;

  (* ---- сброс ошибки команды ---- *)
  StrSw.CommandFault := command_error_for_Status <> 0;
  _errorReset(IN := command_error_for_Status <> 0, PT := T#5S);
  IF _errorReset.Q THEN
  	cmd_for_Status := 0;
  	source_for_Status := 0;
  	command_error_for_Status := 0;
  END_IF;

  outputsSets(in := (StrSw.ISVALIDREF_cmdOn and StrSw.cmdOn ) OR (StrSw.ISVALIDREF_cmdOff and StrSw.cmdOff), PT := T#2S);
  	IF NOT outputsSets.Q THEN
  		StrSw.BreakCmdOn := inBreakCmdOn._inversed AND inBreakCmdOn.reliability AND StrSw.ISVALIDREF_inBreakCmdOn;
  		StrSw.BreakCmdOff := inBreakCmdOff._inversed AND inBreakCmdOff.reliability AND StrSw.ISVALIDREF_inBreakCmdOff;
  	END_IF;

  cmdOn := StrSw.cmdOn;
  cmdOff:= StrSw.cmdOff;

  (* ---- формирование зашифрованного статуса для АРМа ---- *)
  StrSw.status := shl(BYTE_TO_DWORD(source_for_Status), 29)
  		OR shl(BYTE_TO_DWORD(cmd_for_Status), 26)
  		OR shl(BYTE_TO_DWORD(command_error_for_Status), 23)
  		OR shl(bool_to_DWORD(StrSw.sdvig), 22)
  		OR shl(bool_to_DWORD(StrSw.OpcCommandsDisabled), 21)
                      OR shl(bool_to_DWORD(StrSw.lastCmdIsOn), 14)
                      OR shl(BOOL_TO_DWORD(StrSw.BreakCmdOff), 13)
  		OR shl(BOOL_TO_DWORD(StrSw.BreakCmdOn), 12)
                      OR shl(BOOL_TO_DWORD(StrSw.Auto), 7)
  		OR shl(BOOL_TO_DWORD(StrSw.Distance), 6)
  		OR shl(BOOL_TO_DWORD(StrSw.Local), 5)
  		OR shl(BOOL_TO_DWORD(StrSw.Ns), 4)
                  	OR shl(BOOL_TO_DWORD(StrSw.Accident ),3)
  		OR BYTE_TO_DWORD(StrSw.onStatus);
END_FUNCTION_BLOCK

FUNCTION_BLOCK proc_IM
  VAR
    fb_Kran1 : fb_Kran;
    fb_Kran2 : fb_Kran;
    fb_Kran3 : fb_Kran;
    fb_Kran3b : fb_Kran;
    fb_Kran4 : fb_Kran;
    fb_Kran5 : fb_Kran;
    fb_Kran6 : fb_Kran;
    fb_MB : fb_SectionSwitch;
    fb_v1_Avom : fb_Switch;
    fb_v2_Avom : fb_Switch;
    fb_v3_Avom : fb_Switch;
    fb_v4_Avom : fb_Switch;
    fb_Ten_kollect : fb_Switch;
    fb_Ten_MB : fb_Switch;
    fb_pns : fb_Switch;
    fb_nu1 : fb_OilPump;
    fb_nu2 : fb_OilPump;
    fb_Kalorifer_ABO : fb_Switch;
    fb_CMN_pump : fb_Switch;
    fb_PLC_Control : fb_meandr;
  END_VAR
  VAR_EXTERNAL
    di : DiConfig;
    od : DOconfig;
    IM : ImConfig;
  END_VAR
  VAR
    fb_dP_maslo_gaz_menshe_100_kPa : fb_singleSignal;
    fb_dP_gaza_kr_1 : fb_singleSignal;
    fb_otklon_masla_v_akkym_yplot : fb_singleSignal;
    fb_Potok_masla_posle_ABO_bolshe_85_L_min : fb_singleSignal;
    fb_Razreshenie_zagryzki : fb_singleSignal;
    fb_Gotovnosst_vozb : fb_singleSignal;
    fb_Otkl_osn_regylyatora_neisprav : fb_singleSignal;
    fb_ostanov_po_zashitam_vozb_avar : fb_singleSignal;
    fb_SHAVR_1_v_rab : fb_singleSignal;
    fb_SHAVR_2_v_rab : fb_singleSignal;
    fb_Avar_otkl_viklychatelya : fb_singleSignal;
    fb_Asinhron_xod_peregryz : fb_singleSignal;
    fb_AO_KC_ot_SHKC_04M : fb_singleSignal;
    fb_AO_EGPA_ot_PRY : fb_singleSignal;
    fb_EAO_EGPA_ot_PRY : fb_singleSignal;
    fb_Nalichie_220_perem_vhod_v_SHY : fb_singleSignal;
    fb_Nalichie_220_post_vhod_v_SHY : fb_singleSignal;
    fb_Nalichie_220_post_na_shinah_ypr_ZRY : fb_singleSignal;
    fb_BEAO_vkl : fb_singleSignal;
    fb_Net_10_kVt_UcmA_UcmC : fb_singleSignal;
    fb_Net_10_kVt_UcmA_UcmB : fb_singleSignal;
    fb_Srabotka_BREO : fb_singleSignal;
    fb_Sbros_srabotki_BREO : fb_singleSignal;
    fb_NO_GPA_na_SHY : fb_singleSignal;
    fb_AO_GPA_na_SHY : fb_singleSignal;
    fb_EAO_GPA_na_SHY : fb_singleSignal;
    fb_Dver_shkafa_otkrita : fb_singleSignal;
    fb_NKY_vvod_1 : fb_singleSignal;
    fb_NKY_vvod_2 : fb_singleSignal;
    fb_Neisprav_BP_1 : fb_singleSignal;
    fb_Neisprav_BP_2 : fb_singleSignal;
    fb_Neisprav_BP_3 : fb_singleSignal;
    fb_Neisprav_BP_4 : fb_singleSignal;
    fb_Neisprav_BP_5 : fb_singleSignal;
    fb_Neisprav_BP_6 : fb_singleSignal;
    fb_Neisprav_BP_7 : fb_singleSignal;
    fb_Neisprav_BP_8 : fb_singleSignal;
    fb_Neisprav_BP_9 : fb_singleSignal;
    fb_Neisprav_BP_10 : fb_singleSignal;
    fb_Neisprav_cepei_ypr_AVR_pit_vozb : fb_singleSignal;
    fb_Rabota_EGPA : fb_singleOutput;
    fb_Neisparav_EGPA : fb_singleOutput;
    fb_Avar_EGPA : fb_singleOutput;
    fb_Indickaciya_PC_fonar : fb_singleOutput;
    fb_Indickaciya_AC_fonar : fb_singleOutput;
  END_VAR

  (* Циклический опрос. ИМ *)

  (* GPIO *)
  fb_PLC_Control(output:=od.gpio_out.bits[0]);

  (* Кран 1 *)
  fb_Kran1(statOn := di.di_0.bits[1]._inversed, statOn_reliability := di.di_0.bits[1].reliability,
           statOff := di.di_0.bits[0]._inversed, statOff_reliability := di.di_0.bits[0].reliability,
           inSo := di.di_11.bits[0], inSz := di.di_11.bits[1],
           inDp := di.di_2.bits[1],
           cmdOn :=od.do_0.bits[0], cmdOff := od.do_0.bits[1],
           strKr := IM.Kran1  );

    (* Кран 2 *)
  fb_Kran2(statOn := di.di_0.bits[3]._inversed, statOn_reliability:= di.di_0.bits[3].reliability,
           statOff := di.di_0.bits[2]._inversed,  statOff_reliability:= di.di_0.bits[2].reliability,
           inSo := di.di_11.bits[2], inSz := di.di_11.bits[3],
           cmdOn:=od.do_0.bits[3], cmdOff:=od.do_0.bits[4],
           strKr:= IM.Kran2  );

  (* Кран 3 *)
  fb_Kran3(statOn := di.di_0.bits[5]._inversed, statOn_reliability:= di.di_0.bits[5].reliability,
           statOff := di.di_0.bits[4]._inversed,  statOff_reliability:= di.di_0.bits[4].reliability,
           inSo := di.di_11.bits[4], inSz := di.di_11.bits[5],
           cmdOn:=od.do_1.bits[1], cmdOff:=od.do_1.bits[2],
           strKr:= IM.Kran3  );

           (* Кран 3b *)
  fb_Kran3b(statOn := di.di_0.bits[7]._inversed, statOn_reliability:= di.di_0.bits[7].reliability,
           statOff := di.di_0.bits[6]._inversed,  statOff_reliability:= di.di_0.bits[6].reliability,
           inSo := di.di_11.bits[6], inSz := di.di_11.bits[7],
           cmdOn:=od.do_1.bits[3], cmdOff:=od.do_1.bits[4],
           strKr:= IM.Kran3b  );

  (* Кран 4 *)
  fb_Kran4(statOn := di.di_1.bits[1]._inversed, statOn_reliability:= di.di_1.bits[1].reliability,
           statOff := di.di_1.bits[0]._inversed,  statOff_reliability:= di.di_1.bits[0].reliability,
           inSo := di.di_12.bits[0], inSz := di.di_12.bits[1],
           cmdOn:=od.do_2.bits[0], cmdOff:=od.do_2.bits[1],
           strKr:= IM.Kran4  );

  (* Кран 5 *)
  fb_Kran5(statOn := di.di_1.bits[3]._inversed, statOn_reliability:= di.di_1.bits[3].reliability,
           statOff := di.di_1.bits[2]._inversed,  statOff_reliability:= di.di_1.bits[2].reliability,
           inSo := di.di_12.bits[2], inSz := di.di_12.bits[3],
           cmdOn:=od.do_2.bits[2], cmdOff:=od.do_2.bits[3],
           strKr:= IM.Kran5  );

  (* Кран 6 *)
  fb_Kran6(statOn := di.di_1.bits[5]._inversed, statOn_reliability:= di.di_1.bits[5].reliability,
           statOff := di.di_1.bits[4]._inversed,  statOff_reliability:= di.di_1.bits[4].reliability,
           inSo := di.di_12.bits[4], inSz := di.di_12.bits[5],
           cmdOn:=od.do_2.bits[4], cmdOff:=od.do_3.bits[0],
           strKr:= IM.Kran6  );

  (*  MB *)
    fb_MB(statOn := di.di_4.bits[3].value, statOn_reliability:= di.di_4.bits[3].reliability,
           statOff := di.di_4.bits[4].value, statOff_reliability:= di.di_4.bits[4].reliability,
           cmdOn:=od.do_4.bits[0], cmdOff:=od.do_4.bits[1], basketRolledOut := di.di_4.bits[5],
           StrSw:= IM.MB  );

  (*  В1 АВОМ вентилятор охлаждения *)
    fb_v1_Avom(statOn := di.di_5.bits[0].value, statOn_reliability:= di.di_5.bits[0].reliability, inAuto:= di.di_5.bits[2],
           statOff := di.di_5.bits[1].value, statOff_reliability:= di.di_5.bits[1].reliability,
           inBreakCmdOn := di.di_14.bits[2],
           cmdOn:=od.do_5.bits[0] ,
           StrSw:= IM.v1_Avom  );

  (*  В2 АВОМ вентилятор охлаждения *)
    fb_v2_Avom(statOn := di.di_5.bits[3].value, statOn_reliability:= di.di_5.bits[3].reliability, inAuto:= di.di_5.bits[5],
           statOff := di.di_5.bits[4].value, statOff_reliability:= di.di_5.bits[4].reliability,
           inBreakCmdOn := di.di_14.bits[3],
           cmdOn:=od.do_5.bits[1] ,
           StrSw:= IM.v2_Avom  );

    (*  В3 АВОМ вентилятор охлаждения *)
    fb_v3_Avom(statOn := di.di_5.bits[6].value, statOn_reliability:= di.di_5.bits[6].reliability, inAuto:= di.di_6.bits[0],
           statOff := di.di_5.bits[7].value, statOff_reliability:= di.di_5.bits[7].reliability,
           inBreakCmdOn := di.di_14.bits[4],
           cmdOn:=od.do_5.bits[2] ,
           StrSw:= IM.v3_Avom  );

  (*  В4 АВОМ вентилятор охлаждения *)
    fb_v4_Avom(statOn := di.di_6.bits[1].value, statOn_reliability:= di.di_6.bits[1].reliability, inAuto:= di.di_6.bits[3],
           statOff := di.di_6.bits[2].value, statOff_reliability:= di.di_6.bits[2].reliability,
           inBreakCmdOn := di.di_14.bits[5],
           cmdOn:=od.do_5.bits[3] ,
           StrSw:= IM.v4_Avom  );

  (*  ТЭН MB *)
    fb_Ten_MB(statOn := di.di_6.bits[4].value, statOn_reliability:= di.di_6.bits[4].reliability, inAuto:= di.di_6.bits[6],
           statOff := di.di_6.bits[5].value, statOff_reliability:= di.di_6.bits[5].reliability,
           inBreakCmdOn := di.di_14.bits[6],
           cmdOn:=od.do_6.bits[2],
           StrSw:= IM.Ten_MB  );

  (*  ТЭН коллектора *)
    fb_Ten_kollect(statOn := di.di_6.bits[7].value, statOn_reliability:= di.di_7.bits[0].reliability, inAuto:= di.di_7.bits[1],
           statOff := di.di_7.bits[0].value, statOff_reliability:= di.di_7.bits[0].reliability,
           inBreakCmdOn := di.di_14.bits[7],
           cmdOn:=od.do_6.bits[4],
           StrSw:= IM.Ten_kollect  );

    (*  CMN_pump-циркуляционный насос *)
    fb_CMN_pump(statOn := di.di_7.bits[2].value, statOn_reliability:= di.di_7.bits[2].reliability, inAuto:= di.di_7.bits[4],
           statOff := di.di_7.bits[3].value, statOff_reliability:= di.di_7.bits[3].reliability,
           inBreakCmdOn := di.di_15.bits[0],
           cmdOn:=od.do_6.bits[3],
           StrSw:= IM.CMN_pump  );

   (*  ПНС Насос смазки *)
    fb_pns(statOn := di.di_7.bits[5].value, statOn_reliability:= di.di_7.bits[5].reliability, inAuto:= di.di_7.bits[7],
           statOff := di.di_7.bits[6].value, statOff_reliability:= di.di_7.bits[6].reliability,
           inBreakCmdOn := di.di_15.bits[1], cmdOn:=od.do_5.bits[4],
           StrSw:= IM.pns  );

  (*  НУ1  *)
    fb_nu1(statOn := di.di_8.bits[1].value, statOn_reliability:= di.di_8.bits[1].reliability, inAuto:= di.di_8.bits[3],
           statOff := di.di_8.bits[2].value, statOff_reliability:= di.di_8.bits[2].reliability,
           inBreakCmdOn := di.di_15.bits[2], cmdOn:=od.do_6.bits[0],
           StrSw:= IM.nu1  );

  (*  НУ2  *)
    fb_nu2(statOn := di.di_8.bits[4].value, statOn_reliability:= di.di_8.bits[4].reliability, inAuto:= di.di_8.bits[6],
           statOff := di.di_8.bits[5].value, statOff_reliability:= di.di_8.bits[5].reliability,
           inBreakCmdOn := di.di_15.bits[3], cmdOn:=od.do_6.bits[1],
           StrSw:= IM.nu2  );

  (*  Калорифер *)
    fb_Kalorifer_ABO(statOn := di.di_8.bits[7].value, statOn_reliability:= di.di_8.bits[7].reliability, inAuto:= di.di_9.bits[1],
           statOff := di.di_9.bits[0].value, statOff_reliability:= di.di_9.bits[0].reliability,
           inBreakCmdOn := di.di_15.bits[4],
           cmdOn:=od.do_7.bits[0],
           StrSw:= IM.Kalorifer_ABO  );

  (*************************************************** singleSignals ********************************************)

  fb_dP_maslo_gaz_menshe_100_kPa(signal :=di.di_2.bits[0], str_SS :=  IM.SingleSignals.dP_maslo_gaz_menshe_100_kPa);

  fb_dP_gaza_kr_1(signal :=di.di_2.bits[1], str_SS :=  IM.SingleSignals.dP_gaza_kr_1);

  fb_otklon_masla_v_akkym_yplot(signal :=di.di_2.bits[2], str_SS :=  IM.SingleSignals.otklon_masla_v_akkym_yplot);

  fb_Potok_masla_posle_ABO_bolshe_85_L_min(signal :=di.di_2.bits[3], str_SS :=  IM.SingleSignals.Potok_masla_posle_ABO_bolshe_85_L_min);

  fb_Razreshenie_zagryzki(signal :=di.di_3.bits[0], str_SS :=  IM.SingleSignals.Razreshenie_zagryzki);

  fb_Gotovnosst_vozb(signal :=di.di_3.bits[1], str_SS :=  IM.SingleSignals.Gotovnosst_vozb);

  fb_Otkl_osn_regylyatora_neisprav(signal :=di.di_3.bits[2], str_SS :=  IM.SingleSignals.Otkl_osn_regylyatora_neisprav);

  fb_ostanov_po_zashitam_vozb_avar(signal :=di.di_3.bits[3], str_SS :=  IM.SingleSignals.ostanov_po_zashitam_vozb_avar);

  fb_SHAVR_1_v_rab(signal :=di.di_4.bits[1], str_SS :=  IM.SingleSignals.SHAVR_1_v_rab);

  fb_SHAVR_2_v_rab(signal :=di.di_4.bits[2], str_SS :=  IM.SingleSignals.SHAVR_2_v_rab);

  fb_Avar_otkl_viklychatelya(signal :=di.di_4.bits[6], str_SS :=  IM.SingleSignals.Avar_otkl_viklychatelya);

  fb_Asinhron_xod_peregryz(signal :=di.di_4.bits[7], str_SS :=  IM.SingleSignals.Asinhron_xod_peregryz);

  fb_AO_KC_ot_SHKC_04M(signal :=di.di_9.bits[5], str_SS :=  IM.SingleSignals.AO_KC_ot_SHKC_04M);

  fb_AO_EGPA_ot_PRY(signal :=di.di_9.bits[6], str_SS :=  IM.SingleSignals.AO_EGPA_ot_PRY);

  fb_EAO_EGPA_ot_PRY(signal :=di.di_9.bits[7], str_SS :=  IM.SingleSignals.EAO_EGPA_ot_PRY);

  fb_Nalichie_220_perem_vhod_v_SHY(signal :=di.di_13.bits[0], str_SS :=  IM.SingleSignals.Nalichie_220_perem_vhod_v_SHY);

  fb_Nalichie_220_post_vhod_v_SHY(signal :=di.di_13.bits[1], str_SS :=  IM.SingleSignals.Nalichie_220_post_vhod_v_SHY);

  fb_Nalichie_220_post_na_shinah_ypr_ZRY(signal :=di.di_13.bits[2], str_SS :=  IM.SingleSignals.Nalichie_220_post_na_shinah_ypr_ZRY);

  fb_BEAO_vkl(signal :=di.di_16.bits[0], str_SS :=  IM.SingleSignals.BEAO_vkl);

  fb_Net_10_kVt_UcmA_UcmC(signal :=di.di_16.bits[6], str_SS :=  IM.SingleSignals.Net_10_kVt_UcmA_UcmC);

  fb_Net_10_kVt_UcmA_UcmB(signal :=di.di_16.bits[7], str_SS :=  IM.SingleSignals.Net_10_kVt_UcmA_UcmB);

  fb_Srabotka_BREO(signal :=di.di_17.bits[0], str_SS :=  IM.SingleSignals.Srabotka_BREO);

  fb_Sbros_srabotki_BREO(signal :=di.di_17.bits[1], str_SS :=  IM.SingleSignals.Sbros_srabotki_BREO);

  fb_NO_GPA_na_SHY(signal :=di.di_17.bits[4], str_SS :=  IM.SingleSignals.NO_GPA_na_SHY);

  fb_AO_GPA_na_SHY(signal :=di.di_17.bits[5], str_SS :=  IM.SingleSignals.AO_GPA_na_SHY);

  fb_EAO_GPA_na_SHY(signal :=di.di_17.bits[6], str_SS :=  IM.SingleSignals.EAO_GPA_na_SHY);

  fb_Dver_shkafa_otkrita(signal :=di.di_17.bits[7], str_SS :=  IM.SingleSignals.Dver_shkafa_otkrita);

  fb_NKY_vvod_1(signal :=di.di_3.bits[6], str_SS :=  IM.SingleSignals.NKY_vvod_1);

  fb_NKY_vvod_2(signal :=di.di_3.bits[7], str_SS :=  IM.SingleSignals.NKY_vvod_2);

  fb_Neisprav_BP_1(signal :=di.di_10.bits[0], str_SS :=  IM.SingleSignals.Neisprav_BP_1);

  fb_Neisprav_BP_2(signal :=di.di_10.bits[1], str_SS :=  IM.SingleSignals.Neisprav_BP_2);

  fb_Neisprav_BP_3(signal :=di.di_10.bits[2], str_SS :=  IM.SingleSignals.Neisprav_BP_3);

  fb_Neisprav_BP_4(signal :=di.di_10.bits[3], str_SS :=  IM.SingleSignals.Neisprav_BP_4);

  fb_Neisprav_BP_5(signal :=di.di_10.bits[4], str_SS :=  IM.SingleSignals.Neisprav_BP_5);

  fb_Neisprav_BP_6(signal :=di.di_10.bits[5], str_SS :=  IM.SingleSignals.Neisprav_BP_6);

  fb_Neisprav_BP_7(signal :=di.di_10.bits[6], str_SS :=  IM.SingleSignals.Neisprav_BP_7);

  fb_Neisprav_BP_8(signal :=di.di_10.bits[7], str_SS :=  IM.SingleSignals.Neisprav_BP_8);

  fb_Neisprav_BP_9(signal :=di.di_13.bits[3], str_SS :=  IM.SingleSignals.Neisprav_BP_9);

  fb_Neisprav_BP_10(signal :=di.di_13.bits[4], str_SS :=  IM.SingleSignals.Neisprav_BP_10);

  fb_Neisprav_cepei_ypr_AVR_pit_vozb(signal :=di.di_4.bits[0], str_SS :=  IM.SingleSignals.Neisprav_cepei_ypr_AVR_pit_vozb);

  (*************************************************** SingleOutputs ********************************************)

  fb_Rabota_EGPA(str_SO :=  IM.SingleOutputs.Rabota_EGPA,signal:=od.do_8.bits[0]);

  fb_Neisparav_EGPA(str_SO :=  IM.SingleOutputs.Neisparav_EGPA,signal:=od.do_8.bits[1]);

  fb_Avar_EGPA(str_SO :=  IM.SingleOutputs.Avar_EGPA,signal:=od.do_8.bits[2]);

  fb_Indickaciya_PC_fonar(str_SO :=  IM.SingleOutputs.Indickaciya_PC_fonar,signal:=od.do_9.bits[3]);

  fb_Indickaciya_AC_fonar(str_SO :=  IM.SingleOutputs.Indickaciya_AC_fonar,signal:=od.do_9.bits[4]);

   (**************************************** Аналоговые и Дискретные параметры ***********************************)

    (* Гистерезис температуры вклюючения вентиляторов в алгоритме АвтоАВОМ  *)
  (*fb_AutoAvom_hysteresis(StrAP:=IM.AutoAvom_hysteresis);*)

    (* Переключатель разблокировки кранов: 1 - допстить управление кранами  *)
  (*fb_TypeSwitch(StrDP:=IM.TypeSwitch);*)
END_FUNCTION_BLOCK

FUNCTION_BLOCK proc_IM_Init
  VAR
    stOp_Ini : fb_OilPump_Init;
    stSSw_Ini : fb_SectionSwitch_Init;
  END_VAR
  VAR_INPUT
    init : BOOL;
  END_VAR
  VAR
    stKr_Ini : fb_Kran_Init;
    stSw_Ini : fb_Switch_Init;
    stAp_Ini : fb_AnalogParametr_Init;
    stDp_Ini : fb_DiscretParametr_Init;
    stSs_Ini : fb_singleSignal_Init;
    stSo_Ini : fb_singleOutput_Init;
    inits : UINT;
  END_VAR
  VAR_INPUT
    initiales : UINT;
  END_VAR
  VAR_EXTERNAL
    IM : ImConfig;
  END_VAR

  inits := 0; (* Флаг необходимости инициализации структур-дескрипторов *)

                                       (* Стартовая инициализация ИМ *)
  (* Кран 1 *)
  stKr_Ini(data_Ini := true, ISVALIDREF_statOn:=true, ISVALIDREF_statOff:=true,
        ISVALIDREF_cmdOn:=true, ISVALIDREF_cmdOff:=true, ISVALIDREF_inDp:=true,
        ISVALIDREF_inSo:=true, ISVALIDREF_inSz:=true,
        str_Kr := IM.Kran1);
  inits := inits + BOOL_TO_UINT(stKr_Ini.Init);

  (* Кран 2 *)
  stKr_Ini(data_Ini := true, ISVALIDREF_statOn:=true, ISVALIDREF_statOff:=true,
        ISVALIDREF_cmdOn:=true, ISVALIDREF_cmdOff:=true,
        ISVALIDREF_inSo:=true, ISVALIDREF_inSz:=true,
        str_Kr := IM.Kran2);
  inits := inits + BOOL_TO_UINT(stKr_Ini.Init);

  (* Кран 3b *)
  stKr_Ini(data_Ini := true, ISVALIDREF_statOn:=true, ISVALIDREF_statOff:=true,
        ISVALIDREF_cmdOn:=true, ISVALIDREF_cmdOff:=true,
        ISVALIDREF_inSo:=true, ISVALIDREF_inSz:=true, continueHoldCommand:=T#5S,
        str_Kr := IM.Kran3b);
  inits := inits + BOOL_TO_UINT(stKr_Ini.Init);

  (* Кран 4 *)
  stKr_Ini(data_Ini := true, ISVALIDREF_statOn:=true, ISVALIDREF_statOff:=true,
        ISVALIDREF_cmdOn:=true, ISVALIDREF_cmdOff:=true,
        ISVALIDREF_inSo:=true, ISVALIDREF_inSz:=true,
        str_Kr := IM.Kran4);
  inits := inits + BOOL_TO_UINT(stKr_Ini.Init);

  (* Кран 5 *)
  stKr_Ini(data_Ini := true, ISVALIDREF_statOn:=true, ISVALIDREF_statOff:=true,
        ISVALIDREF_cmdOn:=true, ISVALIDREF_cmdOff:=true,
        ISVALIDREF_inSo:=true, ISVALIDREF_inSz:=true,
        str_Kr := IM.Kran5);
  inits := inits + BOOL_TO_UINT(stKr_Ini.Init);

  (* Кран 6 *)
  stKr_Ini(data_Ini := true, ISVALIDREF_statOn:=true, ISVALIDREF_statOff:=true,
        ISVALIDREF_cmdOn:=true, ISVALIDREF_cmdOff:=true,
        ISVALIDREF_inSo:=true, ISVALIDREF_inSz:=true,
        str_Kr := IM.Kran6);
  inits := inits + BOOL_TO_UINT(stKr_Ini.Init);

  (* MB *)
  stSSw_Ini(data_Ini := true, ISVALIDREF_statOn:=true, ISVALIDREF_statOff:=true,
        ISVALIDREF_cmdOn:=true, ISVALIDREF_cmdOff:=true,
        ISVALIDREF_basketRolledOut:=true,
        (*ISVALIDREF_inBreakCmdOn:=true, ISVALIDREF_inBreakCmdOff:=true,*)
        str_Sw := IM.MB);
  inits := inits + BOOL_TO_UINT(stSSw_Ini.Init);

  (* В1 АВОМ вентилятор охлаждения *)
  stSw_Ini(data_Ini := true, ISVALIDREF_statOn:=true, ISVALIDREF_statOff:=true,
        ISVALIDREF_cmdOn:=true,
        ISVALIDREF_inBreakCmdOn:=true, (*ISVALIDREF_inBreakCmdOff:=true,*)
        str_Sw := IM.v1_Avom);
  inits := inits + BOOL_TO_UINT(stSw_Ini.Init);

  (* В2 АВОМ вентилятор охлаждения *)
  stSw_Ini(data_Ini := true, ISVALIDREF_statOn:=true, ISVALIDREF_statOff:=true,
        ISVALIDREF_cmdOn:=true,
        ISVALIDREF_inBreakCmdOn:=true, (*ISVALIDREF_inBreakCmdOff:=true,*)
        str_Sw := IM.v1_Avom);
  inits := inits + BOOL_TO_UINT(stSw_Ini.Init);

  (* В3 АВОМ вентилятор охлаждения *)
  stSw_Ini(data_Ini := true, ISVALIDREF_statOn:=true, ISVALIDREF_statOff:=true,
        ISVALIDREF_cmdOn:=true,
        ISVALIDREF_inBreakCmdOn:=true, (*ISVALIDREF_inBreakCmdOff:=true,*)
        str_Sw := IM.v1_Avom);
  inits := inits + BOOL_TO_UINT(stSw_Ini.Init);

  (* В4 АВОМ вентилятор охлаждения *)
  stSw_Ini(data_Ini := true, ISVALIDREF_statOn:=true, ISVALIDREF_statOff:=true,
        ISVALIDREF_cmdOn:=true,
        ISVALIDREF_inBreakCmdOn:=true,(*ISVALIDREF_inBreakCmdOff:=true,*)
        str_Sw := IM.v1_Avom);
  inits := inits + BOOL_TO_UINT(stSw_Ini.Init);

  (* ТЭН маслобака *)
  stSw_Ini(data_Ini := true, ISVALIDREF_statOn:=true, ISVALIDREF_statOff:=true,
        ISVALIDREF_cmdOn:=true,
        ISVALIDREF_inBreakCmdOn:=true,
        str_Sw := IM.Ten_MB);
  inits := inits + BOOL_TO_UINT(stSw_Ini.Init);

  (* ТЭН коллектора *)
  stSw_Ini(data_Ini := true, ISVALIDREF_statOn:=true, ISVALIDREF_statOff:=true,
        ISVALIDREF_cmdOn:=true,
        ISVALIDREF_inBreakCmdOn:=true,
        str_Sw := IM.Ten_kollect);
  inits := inits + BOOL_TO_UINT(stSw_Ini.Init);

  (* CMN_pump-циркуляционный насос *)
  stSw_Ini(data_Ini := true, ISVALIDREF_statOn:=true, ISVALIDREF_statOff:=true,
        ISVALIDREF_cmdOn:=true,
        ISVALIDREF_inBreakCmdOn:=true,
        str_Sw := IM.CMN_pump);
  inits := inits + BOOL_TO_UINT(stSw_Ini.Init);

  (* ПНС Насос смазки *)
  stSw_Ini(data_Ini := true, ISVALIDREF_statOn:=true, ISVALIDREF_statOff:=true,
        ISVALIDREF_cmdOn:=true,
        ISVALIDREF_inBreakCmdOn:=true,
       (*ISVALIDREF_inBreakCmdOff:=true,*)
        str_Sw := IM.pns);
  inits := inits + BOOL_TO_UINT(stSw_Ini.Init);

  (* nu1 *)
  stOp_Ini(data_Ini := true, ISVALIDREF_statOn:=true, ISVALIDREF_statOff:=true,
        ISVALIDREF_cmdOn:=true,
        ISVALIDREF_inBreakCmdOn:=true,
        str_Op := IM.nu1);
  inits := inits + BOOL_TO_UINT(stOp_Ini.Init);

  (* nu2 *)
  stOp_Ini(data_Ini := true, ISVALIDREF_statOn:=true, ISVALIDREF_statOff:=true,
        ISVALIDREF_cmdOn:=true,
        ISVALIDREF_inBreakCmdOn:=true,
        str_Op := IM.nu2);
  inits := inits + BOOL_TO_UINT(stOp_Ini.Init);

                                                          (* Стартовая инициализация singleSignal *)

  (* dP_maslo_gaz_menshe_100_kPa *)
  stSs_Ini(data_Ini := true, inverse:=FALSE, (*DelayOn:=T#0S, DelayOff:=T#0S,*) str_SS := IM.SingleSignals.dP_maslo_gaz_menshe_100_kPa);
  inits := inits + BOOL_TO_UINT(stSs_Ini.Init);

  (* dP_gaza_kr_1 *)
  stSs_Ini(data_Ini := true, inverse:=FALSE, (*DelayOn:=T#0S, DelayOff:=T#0S,*) str_SS := IM.SingleSignals.dP_gaza_kr_1);
  inits := inits + BOOL_TO_UINT(stSs_Ini.Init);

  (* otklon_masla_v_akkym_yplot *)
  stSs_Ini(data_Ini := true, inverse:=FALSE, (*DelayOn:=T#0S, DelayOff:=T#0S,*) str_SS := IM.SingleSignals.otklon_masla_v_akkym_yplot);
  inits := inits + BOOL_TO_UINT(stSs_Ini.Init);

  (* Potok_masla_posle_ABO_bolshe_85_L_min *)
  stSs_Ini(data_Ini := true, inverse:=TRUE, (*DelayOn:=T#0S, DelayOff:=T#0S,*) str_SS := IM.SingleSignals.Potok_masla_posle_ABO_bolshe_85_L_min);
  inits := inits + BOOL_TO_UINT(stSs_Ini.Init);

  (* Razreshenie_zagryzki *)
  stSs_Ini(data_Ini := true, inverse:=FALSE, (*DelayOn:=T#0S, DelayOff:=T#0S,*) str_SS := IM.SingleSignals.Razreshenie_zagryzki);
  inits := inits + BOOL_TO_UINT(stSs_Ini.Init);

  (* Gotovnosst_vozb *)
  stSs_Ini(data_Ini := true, inverse:=FALSE, (*DelayOn:=T#0S, DelayOff:=T#0S,*) str_SS := IM.SingleSignals.Gotovnosst_vozb);
  inits := inits + BOOL_TO_UINT(stSs_Ini.Init);

  (* Otkl_osn_regylyatora_neisprav *)
  stSs_Ini(data_Ini := true, inverse:=FALSE, (*DelayOn:=T#0S, DelayOff:=T#0S,*) str_SS := IM.SingleSignals.Otkl_osn_regylyatora_neisprav);
  inits := inits + BOOL_TO_UINT(stSs_Ini.Init);

  (* ostanov_po_zashitam_vozb_avar *)
  stSs_Ini(data_Ini := true, inverse:=FALSE, (*DelayOn:=T#0S, DelayOff:=T#0S,*) str_SS := IM.SingleSignals.ostanov_po_zashitam_vozb_avar);
  inits := inits + BOOL_TO_UINT(stSs_Ini.Init);

  (* NKY_vvod_1 *)
  stSs_Ini(data_Ini := true, inverse:=FALSE, (*DelayOn:=T#0S, DelayOff:=T#0S,*) str_SS := IM.SingleSignals.NKY_vvod_1);
  inits := inits + BOOL_TO_UINT(stSs_Ini.Init);

  (* NKY_vvod_2 *)
  stSs_Ini(data_Ini := true, inverse:=FALSE, (*DelayOn:=T#0S, DelayOff:=T#0S,*) str_SS := IM.SingleSignals.NKY_vvod_2);
  inits := inits + BOOL_TO_UINT(stSs_Ini.Init);

  (* Neisprav_cepei_ypr_AVR_pit_vozb *)
  stSs_Ini(data_Ini := true, inverse:=TRUE, (*DelayOn:=T#0S, DelayOff:=T#0S,*) str_SS := IM.SingleSignals.Neisprav_cepei_ypr_AVR_pit_vozb);
  inits := inits + BOOL_TO_UINT(stSs_Ini.Init);

  (* SHAVR_1_v_rab *)
  stSs_Ini(data_Ini := true, inverse:=FALSE, (*DelayOn:=T#0S, DelayOff:=T#0S,*) str_SS := IM.SingleSignals.SHAVR_1_v_rab);
  inits := inits + BOOL_TO_UINT(stSs_Ini.Init);

  (* SHAVR_2_v_rab *)
  stSs_Ini(data_Ini := true, inverse:=FALSE, (*DelayOn:=T#0S, DelayOff:=T#0S,*) str_SS := IM.SingleSignals.SHAVR_2_v_rab);
  inits := inits + BOOL_TO_UINT(stSs_Ini.Init);

  (* Avar_otkl_viklychatelya *)
  stSs_Ini(data_Ini := true, inverse:=FALSE, (*DelayOn:=T#0S, DelayOff:=T#0S,*) str_SS := IM.SingleSignals.Avar_otkl_viklychatelya);
  inits := inits + BOOL_TO_UINT(stSs_Ini.Init);

  (* Asinhron_xod_peregryz *)
  stSs_Ini(data_Ini := true, inverse:=FALSE, (*DelayOn:=T#0S, DelayOff:=T#0S,*) str_SS := IM.SingleSignals.Asinhron_xod_peregryz);
  inits := inits + BOOL_TO_UINT(stSs_Ini.Init);

  (* AO_KC_ot_SHKC_04M *)
  stSs_Ini(data_Ini := true, inverse:=FALSE, (*DelayOn:=T#0S, DelayOff:=T#0S,*) str_SS := IM.SingleSignals.AO_KC_ot_SHKC_04M);
  inits := inits + BOOL_TO_UINT(stSs_Ini.Init);

  (* AO_EGPA_ot_PRY *)
  stSs_Ini(data_Ini := true, inverse:=FALSE, (*DelayOn:=T#0S, DelayOff:=T#0S,*) str_SS := IM.SingleSignals.AO_EGPA_ot_PRY);
  inits := inits + BOOL_TO_UINT(stSs_Ini.Init);

  (* EAO_EGPA_ot_PRY *)
  stSs_Ini(data_Ini := true, inverse:=FALSE, (*DelayOn:=T#0S, DelayOff:=T#0S,*) str_SS := IM.SingleSignals.EAO_EGPA_ot_PRY);
  inits := inits + BOOL_TO_UINT(stSs_Ini.Init);

  (* Nalichie_220_perem_vhod_v_SHY *)
  stSs_Ini(data_Ini := true, inverse:=FALSE, (*DelayOn:=T#0S, DelayOff:=T#0S,*) str_SS := IM.SingleSignals.Nalichie_220_perem_vhod_v_SHY);
  inits := inits + BOOL_TO_UINT(stSs_Ini.Init);

  (* Nalichie_220_post_vhod_v_SHY *)
  stSs_Ini(data_Ini := true, inverse:=FALSE, (*DelayOn:=T#0S, DelayOff:=T#0S,*) str_SS := IM.SingleSignals.Nalichie_220_post_vhod_v_SHY);
  inits := inits + BOOL_TO_UINT(stSs_Ini.Init);

  (* Nalichie_220_post_na_shinah_ypr_ZRY *)
  stSs_Ini(data_Ini := true, inverse:=FALSE, (*DelayOn:=T#0S, DelayOff:=T#0S,*) str_SS := IM.SingleSignals.Nalichie_220_post_na_shinah_ypr_ZRY);
  inits := inits + BOOL_TO_UINT(stSs_Ini.Init);

  (* BEAO_vkl *)
  stSs_Ini(data_Ini := true, inverse:=FALSE, (*DelayOn:=T#0S, DelayOff:=T#0S,*) str_SS := IM.SingleSignals.BEAO_vkl);
  inits := inits + BOOL_TO_UINT(stSs_Ini.Init);

  (* Net_10_kVt_UcmA_UcmC *)
  stSs_Ini(data_Ini := true, inverse:=FALSE, (*DelayOn:=T#0S, DelayOff:=T#0S,*) str_SS := IM.SingleSignals.Net_10_kVt_UcmA_UcmC);
  inits := inits + BOOL_TO_UINT(stSs_Ini.Init);

  (* Net_10_kVt_UcmA_UcmB *)
  stSs_Ini(data_Ini := true, inverse:=FALSE, (*DelayOn:=T#0S, DelayOff:=T#0S,*) str_SS := IM.SingleSignals.Net_10_kVt_UcmA_UcmB);
  inits := inits + BOOL_TO_UINT(stSs_Ini.Init);

  (* Srabotka_BREO *)
  stSs_Ini(data_Ini := true, inverse:=FALSE, (*DelayOn:=T#0S, DelayOff:=T#0S,*) str_SS := IM.SingleSignals.Srabotka_BREO);
  inits := inits + BOOL_TO_UINT(stSs_Ini.Init);

  (* Sbros_srabotki_BREO *)
  stSs_Ini(data_Ini := true, inverse:=FALSE, (*DelayOn:=T#0S, DelayOff:=T#0S,*) str_SS := IM.SingleSignals.Sbros_srabotki_BREO);
  inits := inits + BOOL_TO_UINT(stSs_Ini.Init);

  (* NO_GPA_na_SHY *)
  stSs_Ini(data_Ini := true, inverse:=FALSE, (*DelayOn:=T#0S, DelayOff:=T#0S,*) str_SS := IM.SingleSignals.NO_GPA_na_SHY);
  inits := inits + BOOL_TO_UINT(stSs_Ini.Init);

  (* AO_GPA_na_SHY *)
  stSs_Ini(data_Ini := true, inverse:=FALSE, (*DelayOn:=T#0S, DelayOff:=T#0S,*) str_SS := IM.SingleSignals.AO_GPA_na_SHY);
  inits := inits + BOOL_TO_UINT(stSs_Ini.Init);

  (* EAO_GPA_na_SHY *)
  stSs_Ini(data_Ini := true, inverse:=FALSE, (*DelayOn:=T#0S, DelayOff:=T#0S,*) str_SS := IM.SingleSignals.EAO_GPA_na_SHY);
  inits := inits + BOOL_TO_UINT(stSs_Ini.Init);

  (* Dver_shkafa_otkrita *)
  stSs_Ini(data_Ini := true, inverse:=TRUE, (*DelayOn:=T#0S, DelayOff:=T#0S,*) str_SS := IM.SingleSignals.Dver_shkafa_otkrita);
  inits := inits + BOOL_TO_UINT(stSs_Ini.Init);

  (* Neisprav_BP_1 *)
  stSs_Ini(data_Ini := true, inverse:=FALSE, (*DelayOn:=T#0S, DelayOff:=T#0S,*) str_SS := IM.SingleSignals.Neisprav_BP_1);
  inits := inits + BOOL_TO_UINT(stSs_Ini.Init);

  (* Neisprav_BP_2 *)
  stSs_Ini(data_Ini := true, inverse:=FALSE, (*DelayOn:=T#0S, DelayOff:=T#0S,*) str_SS := IM.SingleSignals.Neisprav_BP_2);
  inits := inits + BOOL_TO_UINT(stSs_Ini.Init);

  (* Neisprav_BP_3 *)
  stSs_Ini(data_Ini := true, inverse:=FALSE, (*DelayOn:=T#0S, DelayOff:=T#0S,*) str_SS := IM.SingleSignals.Neisprav_BP_3);
  inits := inits + BOOL_TO_UINT(stSs_Ini.Init);

  (* Neisprav_BP_4 *)
  stSs_Ini(data_Ini := true, inverse:=FALSE, (*DelayOn:=T#0S, DelayOff:=T#0S,*) str_SS := IM.SingleSignals.Neisprav_BP_4);
  inits := inits + BOOL_TO_UINT(stSs_Ini.Init);

  (* Neisprav_BP_5 *)
  stSs_Ini(data_Ini := true, inverse:=FALSE, (*DelayOn:=T#0S, DelayOff:=T#0S,*) str_SS := IM.SingleSignals.Neisprav_BP_5);
  inits := inits + BOOL_TO_UINT(stSs_Ini.Init);

  (* Neisprav_BP_6 *)
  stSs_Ini(data_Ini := true, inverse:=FALSE, (*DelayOn:=T#0S, DelayOff:=T#0S,*) str_SS := IM.SingleSignals.Neisprav_BP_6);
  inits := inits + BOOL_TO_UINT(stSs_Ini.Init);

  (* Neisprav_BP_7 *)
  stSs_Ini(data_Ini := true, inverse:=FALSE, (*DelayOn:=T#0S, DelayOff:=T#0S,*) str_SS := IM.SingleSignals.Neisprav_BP_7);
  inits := inits + BOOL_TO_UINT(stSs_Ini.Init);

  (* Neisprav_BP_8 *)
  stSs_Ini(data_Ini := true, inverse:=FALSE, (*DelayOn:=T#0S, DelayOff:=T#0S,*) str_SS := IM.SingleSignals.Neisprav_BP_8);
  inits := inits + BOOL_TO_UINT(stSs_Ini.Init);

  (* Neisprav_BP_9 *)
  stSs_Ini(data_Ini := true, inverse:=FALSE, (*DelayOn:=T#0S, DelayOff:=T#0S,*) str_SS := IM.SingleSignals.Neisprav_BP_9);
  inits := inits + BOOL_TO_UINT(stSs_Ini.Init);

  (* Neisprav_BP_10 *)
  stSs_Ini(data_Ini := true, inverse:=FALSE, (*DelayOn:=T#0S, DelayOff:=T#0S,*) str_SS := IM.SingleSignals.Neisprav_BP_10);
  inits := inits + BOOL_TO_UINT(stSs_Ini.Init);

                                      (* Стартовая инициализация singleOutput *)

  (* Rabota_EGPA *)
  stSo_Ini(data_Ini := true, inOpcCommandsDisabled:=FALSE, (*DelayOn:=T#0S, DelayOff:=T#0S,*) str_SO := IM.SingleOutputs.Rabota_EGPA);
  inits := inits + BOOL_TO_UINT(stSo_Ini.Init);

  (* Neisparav_EGPA *)
  stSo_Ini(data_Ini := true, inOpcCommandsDisabled:=TRUE, (*DelayOn:=T#0S, DelayOff:=T#0S,*) str_SO := IM.SingleOutputs.Neisparav_EGPA);
  inits := inits + BOOL_TO_UINT(stSo_Ini.Init);

  (* Avar_EGPA *)
  stSo_Ini(data_Ini := true, inOpcCommandsDisabled:=FALSE, (*DelayOn:=T#0S, DelayOff:=T#0S,*) str_SO := IM.SingleOutputs.Avar_EGPA);
  inits := inits + BOOL_TO_UINT(stSo_Ini.Init);

  (* Indickaciya_PC_fonar *)
  stSo_Ini(data_Ini := true, inOpcCommandsDisabled:=FALSE, (*DelayOn:=T#0S, DelayOff:=T#0S,*) str_SO := IM.SingleOutputs.Indickaciya_PC_fonar);
  inits := inits + BOOL_TO_UINT(stSo_Ini.Init);

  (* Indickaciya_AC_fonar *)
  stSo_Ini(data_Ini := true, inOpcCommandsDisabled:=FALSE, (*DelayOn:=T#0S, DelayOff:=T#0S,*) str_SO := IM.SingleOutputs.Indickaciya_AC_fonar);
  inits := inits + BOOL_TO_UINT(stSo_Ini.Init);

  initiales := 0;
  IF init THEN initiales := inits; END_IF;
END_FUNCTION_BLOCK

FUNCTION_BLOCK NOAlg
  VAR_IN_OUT
    StrAlg : struct_Alg;
  END_VAR
  VAR
    sbrosVibeg : struct_Question;
    fb_sbrosVibeg : fb_Question;
    pusk_v : fb_AlgoritmsManager;
    timer120 : struct_PhaseAlgoritm;
    runUnsuccessful : struct_PhaseAlgoritm;
    kran6Open : struct_PhaseAlgoritm;
    kran3bOpen : struct_PhaseAlgoritm;
    MBOff : struct_PhaseAlgoritm;
    kran1Close : struct_PhaseAlgoritm;
    kran2Close : struct_PhaseAlgoritm;
    kran3Close : struct_PhaseAlgoritm;
    kran4Close : struct_PhaseAlgoritm;
    kran5Open : struct_PhaseAlgoritm;
    error_Krans : struct_PhaseAlgoritm;
    autoPnsOff : struct_PhaseAlgoritm;
    pnsOn : struct_PhaseAlgoritm;
    Pg_VhodLessThen300 : struct_PhaseAlgoritm;
    Pg_VyhodLessThen300 : struct_PhaseAlgoritm;
    nu1Off : struct_PhaseAlgoritm;
    nu2Off : struct_PhaseAlgoritm;
    autoNuOff : struct_PhaseAlgoritm;
    timer600 : struct_PhaseAlgoritm;
    Avom1Off : struct_PhaseAlgoritm;
    Avom2Off : struct_PhaseAlgoritm;
    Avom3Off : struct_PhaseAlgoritm;
    Avom4Off : struct_PhaseAlgoritm;
    autoAVOMOff : struct_PhaseAlgoritm;
    timer5 : struct_PhaseAlgoritm;
    fb_timer120 : fb_ph_Timer;
    fb_kran6Open : fb_ph_Kran;
    fb_kran4Close : fb_ph_Kran;
    fb_kran3bOpen : fb_ph_Kran;
    fb_MBOff : fb_ph_SectionSwitch;
    fb_kran1Close : fb_ph_Kran;
    fb_kran2Close : fb_ph_Kran;
    fb_kran3Close : fb_ph_Kran;
    fb_kran5Open : fb_ph_Kran;
    fb_error_Krans : fb_ph_CustomPhase;
    fb_runUnsuccessful : fb_ph_CustomPhase;
    fb_autoPnsOff : fb_ph_algoritm;
    fb_pnsOn : fb_ph_Switch;
    fb_Pg_VhodLessThen300 : fb_ph_CustomPhase;
    fb_Pg_VyhodLessThen300 : fb_ph_CustomPhase;
    fb_nu1Off : fb_ph_OilPump;
    fb_nu2Off : fb_ph_OilPump;
    fb_autoNuOff : fb_ph_Switch;
    fb_timer600 : fb_ph_Timer;
    fb_Avom1Off : fb_ph_Switch;
    fb_Avom2Off : fb_ph_Switch;
    fb_Avom3Off : fb_ph_Switch;
    fb_Avom4Off : fb_ph_Switch;
    fb_autoAVOMOff : fb_ph_algoritm;
    fb_timer5 : fb_ph_Timer;
    _sunpackerCommand : fb_sunpackerCommand;
    _statusAi : TYPE_StatusAi;
    _Answers : TYPE_Answers;
    _statusDualInput : TYPE_statusDualInput;
    _commandDualInput : TYPE_commandDualInput;
    _DualStateImAction : TYPE_DualStateImAction;
    _PhaseAlgoritmAction : TYPE_PhaseAlgoritmAction;
    source : BYTE;
    cmd : BYTE;
    lastCmd : BYTE;
    source_for_Status : BYTE;
    cmd_for_Status : BYTE;
    command_error_for_Status : BYTE;
    resetCmdTimer : TON;
    resetCmdTimerPriznak : BOOL;
    onInit : BOOL;
    waitReset : TON;
  END_VAR
  VAR_EXTERNAL
    IM : ImConfig;
    algoritms : AlgoritmsConfig;
    ai : AiConfig;
    protections : ProtectionsConfig;
    ModeGpa : TYPE_ModeGpa;
    algmanager : struct_AlgoritmsManager;
    AlgTimers : struct_AlgTimers;
  END_VAR
  VAR CONSTANT
    Ust_Pgaza : LREAL      := 0.3;
  END_VAR

  IF NOT onInit THEN

         fb_timer120(phaseNumber:=1);
              fb_kran6Open(phaseNumber:=2, act:=_off);
              fb_kran4Close(phaseNumber:=3, act:=_on);
         fb_kran3bOpen(phaseNumber:=4, act:=_on);
         fb_MBOff(phaseNumber:=5, act:=_off);
         fb_kran1Close(phaseNumber:=6, act:=_off);
          fb_kran2Close(phaseNumber:=7, act:=_on);
          fb_kran3Close(phaseNumber:=8, act:=_off);
         fb_kran5Open(phaseNumber:=9, act:=_off);
      fb_error_Krans(phaseNumber:=10);
        fb_pnsOn(phaseNumber:=11, act:=_on);
        fb_Pg_VhodLessThen300(phaseNumber:=12);
        fb_Pg_VyhodLessThen300(phaseNumber:=13);
             fb_nu1Off(phaseNumber:=14, act:=_off);
             fb_nu2Off(phaseNumber:=15, act:=_off);
             fb_autoNuOff(phaseNumber:=16, act:=_off);
      fb_timer600(phaseNumber:=17, delay:=T#240S);
         fb_Avom1Off(phaseNumber:=18, act:=_off);
         fb_Avom2Off(phaseNumber:=19, act:=_off);
         fb_Avom3Off(phaseNumber:=20, act:=_off);
         fb_Avom4Off(phaseNumber:=21, act:=_off);
         fb_autoAVOMOff(phaseNumber:=22, act:=_reset);
         fb_timer5(phaseNumber:=23);
         fb_runUnsuccessful(phaseNumber:=24);
         fb_sbrosVibeg(phaseNumber:=25);
         (*fb_klapan1(phaseNumber:=24, act:=_run, waitCompletion:=TRUE);
    fb_klapan2(phaseNumber:=25);*)

  onInit:=TRUE;
  END_IF;

         fb_timer120(StrPh:=timer120);
  fb_kran6Open(StrPh:=kran6Open, Im:=Im.kran6);
  fb_kran4Close(StrPh:=kran4Close, Im:=Im.kran4);
  fb_kran3bOpen(StrPh:=kran3bOpen, Im:=Im.kran3b);
  fb_MBOff(StrPh:=MBOff, Im:=Im.MB);
  fb_kran1Close(StrPh:=kran1Close, Im:=Im.kran1);
  fb_kran2Close(StrPh:=kran2Close, Im:=Im.kran2);
  fb_kran3Close(StrPh:=kran3Close, Im:=Im.kran3);
  fb_kran5Open(StrPh:=kran5Open, Im:=Im.kran5);
  fb_error_Krans(StrPh:=error_Krans);
  fb_pnsOn(StrPh:=pnsOn, Im:=Im.pns);
  fb_Pg_VhodLessThen300(StrPh:=Pg_VhodLessThen300);
  fb_Pg_VyhodLessThen300(StrPh:=Pg_VyhodLessThen300);
  fb_nu1Off(StrPh:=nu1Off, Im:=Im.nu1);
  fb_nu2Off(StrPh:=nu2Off, Im:=Im.nu2);
  fb_autoNuOff(StrPh:=autoNuOff);
  fb_timer600(StrPh:=timer600);
  fb_Avom1Off(StrPh:=Avom1Off, Im:=Im.v1_Avom);
  fb_Avom2Off(StrPh:=Avom2Off, Im:=Im.v2_Avom);
  fb_Avom3Off(StrPh:=Avom3Off, Im:=Im.v3_Avom);
  fb_Avom4Off(StrPh:=Avom4Off, Im:=Im.v4_Avom);
  fb_autoAVOMOff(StrPh:=autoAVOMOff);
  fb_timer5(StrPh:=timer5);
  fb_runUnsuccessful(StrPh:=runUnsuccessful);
  fb_sbrosVibeg(strQ:=sbrosVibeg);
  (*fb_klapan1(StrPh:=klapan1, Im:=Im.klapan1);
  fb_klapan2(StrPh:=klapan2, Im:=Im.klapan2);*)

  StrAlg.CanRun := StrAlg.inCanRun;
  StrAlg.OpcCommandsDisabled := StrAlg.inOpcCommandsDisabled;

  IF StrAlg.isRuning THEN

       StrAlg.hasError := kran4Close.error OR MBOff.error OR pnsOn.error OR kran3bOpen.error
      OR kran1Close.error OR kran2Close.error OR kran5Open.error OR kran6Open.error OR runUnsuccessful.error;

      sbrosVibeg.AnswerVariants:=_Answers.ANS_YES;

      IF timer120.top AND NOT kran6Open.top THEN
         runUnsuccessful.error:=TRUE;
      END_IF;
      IF kran6Open.top THEN
          runPhase(kran3bOpen);
      END_IF;
      IF kran3bOpen.top THEN
          runPhase(MBOff);
      END_IF;
      IF MBOff.top THEN
          runPhase(pnsOn);
          runPhase(autoPnsOff);
          runPhase(kran1Close);
          runPhase(kran2Close);
          runPhase(kran3Close);
      END_IF;
      IF kran1Close.top AND kran2Close.top AND kran3Close.top AND kran4Close.top THEN
          runPhase(kran5Open);
      END_IF;
      IF kran5Open.top AND pnsOn.top (*AND pr na vih <300 AND pr na vh < 300*) THEN
          runPhase(nu1Off);
          runPhase(nu2Off);
      END_IF;
      IF nu1Off.top AND nu2Off.top AND NOT algmanager.puskV THEN
          askQuestion(sbrosVibeg);
          runPhase(timer600);
          runPhase(Avom1Off);
          runPhase(Avom2Off);
          runPhase(Avom3Off);
          runPhase(Avom4Off);
          runPhase(autoAVOMOff);
      END_IF;
      IF nu1Off.top AND nu2Off.top AND algmanager.puskV=TRUE THEN
          askQuestion(sbrosVibeg);
          runPhase(Avom1Off);
          runPhase(Avom2Off);
          runPhase(Avom3Off);
          runPhase(Avom4Off);
          runPhase(autoAVOMOff);
      END_IF;
      IF NOT pnsOn.top AND Avom1Off.top AND Avom2Off.top AND Avom3Off.top AND Avom4Off.top AND autoAVOMOff.top THEN
          runPhase(timer5);
      END_IF;
      StrAlg.isEnded:= Avom1Off.top AND Avom2Off.top AND Avom3Off.top AND Avom4Off.top AND NOT pnsOn.top AND autoAVOMOff.top;

  END_IF;

  StrAlg.CanRun := StrAlg.inCanRun;
  StrAlg.OpcCommandsDisabled := StrAlg.inOpcCommandsDisabled;

  (* ---- Если управление с ВУ заблокировано, то  передаем команду из алгоритма ---- *)
  IF StrAlg.inOpcCommandsDisabled THEN
  	StrAlg.inCommand := StrAlg.inCommand_Alg;
  ELSE (* иначе передаем команду с АРМа*)
  	StrAlg.inCommand := StrAlg.inCommand_ARM;
  END_IF;

  _sunpackerCommand(command := StrAlg.inCommand);
  	source := _sunpackerCommand.source;
  	cmd := _sunpackerCommand.cmd;

  IF cmd <> 0 AND lastCmd <> cmd AND (((NOT StrAlg.opcCommandsDisabled) AND source > 0) OR source = 0) then
  	CASE BYTE_TO_INT(cmd) OF
  		(*cmdRun*) 1: 	IF (StrAlg.CanRun) THEN
  					StrAlg.isRuning := TRUE;
  					StrAlg.isEnded := FALSE;
  					StrAlg.hasError := FALSE;
  					(*****************       OnRun       *****************)

                                                    algManager.nMode:=ModeGpa.MODE_NO;

                                                    runPhase(kran6Open);
                                                    runPhase(kran4Close);
                                                    runPhase(timer120);
                                                    runPhase(runUnsuccessful);

                                                    resetAiProtection(protections.Vibroskorost_OP_ED_t1_HA);
                                                    resetAiProtection(protections.Vibroskorost_OYP_ED_so_storony_redyctora_t2_HA);
                                                    resetAiProtection(protections.Vibroskorost_OYP_kolesa_ED_t3_HA);
                                                    resetAiProtection(protections.Vibroskorost_OP_shesterni_nagnetatelya_t6_HA);
                                                    resetDiProtection(protections.Kran1sdvig);
                                                    resetDiProtection(protections.Kran2sdvig);

  					cmd_for_Status := cmd;
  					source_for_Status := source;
  					command_error_for_Status := 0;
  				ELSE
  					StrAlg.isRuning := FALSE;
  					StrAlg.isEnded := FALSE;
  					StrAlg.hasError 	:= FALSE;

  					cmd_for_Status := 0;
  					source_for_Status := source;
  					command_error_for_Status := cmd;
  				END_IF;
  		(*cmdReset*) 2: 	StrAlg.isRuning := FALSE;
  				StrAlg.isEnded := FALSE;
  				StrAlg.hasError 	:= FALSE;

                                           (*****************       OnReset       *****************)
                                          waitReset(IN:=FALSE);
                                          resetIfRunning(algoritms.vibegPNS);

  resetPhase(timer120);
  resetPhase(kran6Open);
  resetPhase(kran4Close);
  resetPhase(kran3bOpen);
  resetPhase(MBOff);
  resetPhase(kran1Close);
  resetPhase(kran2Close);
  resetPhase(kran3Close);
  resetPhase(kran5Open);
  resetPhase(error_Krans);
  resetPhase(pnsOn);
  resetPhase(Pg_VhodLessThen300);
  resetPhase(Pg_VyhodLessThen300);
  resetPhase(nu1Off);
  resetPhase(nu2Off);
  resetPhase(autoNuOff);
  resetPhase(timer600);
  resetPhase(Avom1Off);
  resetPhase(Avom2Off);
  resetPhase(Avom3Off);
  resetPhase(Avom4Off);
  resetPhase(autoAVOMOff);
  resetPhase(timer5);
  resetPhase(runUnsuccessful);
  resetQuestion(sbrosVibeg);
  (*resetPhase(klapan1);
  resetPhase(klapan2);*)

  				cmd_for_Status := cmd;
  				source_for_Status := source;
  				command_error_for_Status := 0;
  	END_CASE;
  	resetCmdTimer(IN := false);
  	resetCmdTimerPriznak := TRUE;
  END_IF;
  lastCmd := cmd;

  resetCmdTimer(IN := resetCmdTimerPriznak, PT := T#5S);
  IF resetCmdTimer.Q THEN
  	resetCmdTimerPriznak := FALSE;
  	source_for_Status := 0;
  	cmd_for_Status := 0;
  	command_error_for_Status := 0;
  END_IF;

  StrAlg.Start:= timer120.startStatus
  OR kran6Open.startStatus
  OR kran4Close.startStatus
  OR kran3bOpen.startStatus
  OR MBOff.startStatus
  OR kran1Close.startStatus
  OR kran2Close.startStatus
  OR kran3Close.startStatus
  OR kran5Open.startStatus
  OR error_Krans.startStatus
  OR pnsOn.startStatus
  OR Pg_VhodLessThen300.startStatus
  OR Pg_VyhodLessThen300.startStatus
  OR nu1Off.startStatus
  OR nu2Off.startStatus
  OR autoNuOff.startStatus
  OR timer600.startStatus
  OR Avom1Off.startStatus
  OR Avom2Off.startStatus
  OR Avom3Off.startStatus
  OR Avom4Off.startStatus
  OR autoAVOMOff.startStatus
  OR timer5.startStatus
  OR runUnsuccessful.startStatus;
  (*OR klapan1.startStatus
  OR klapan2.startStatus;*)

  StrAlg.Error:= timer120.errorStatus
  OR kran6Open.errorStatus
  OR kran4Close.errorStatus
  OR kran3bOpen.errorStatus
  OR MBOff.errorStatus
  OR kran1Close.errorStatus
  OR kran2Close.errorStatus
  OR kran3Close.errorStatus
  OR kran5Open.errorStatus
  OR error_Krans.errorStatus
  OR pnsOn.errorStatus
  OR Pg_VhodLessThen300.errorStatus
  OR Pg_VyhodLessThen300.errorStatus
  OR nu1Off.errorStatus
  OR nu2Off.errorStatus
  OR autoNuOff.errorStatus
  OR timer600.errorStatus
  OR Avom1Off.errorStatus
  OR Avom2Off.errorStatus
  OR Avom3Off.errorStatus
  OR Avom4Off.errorStatus
  OR autoAVOMOff.errorStatus
  OR timer5.errorStatus
  OR runUnsuccessful.errorStatus;
  (*OR klapan1.errorStatus
  OR klapan2.errorStatus;*)

  StrAlg.Top:=   timer120.topStatus
  OR kran6Open.topStatus
  OR kran4Close.topStatus
  OR kran3bOpen.topStatus
  OR MBOff.topStatus
  OR kran1Close.topStatus
  OR kran2Close.topStatus
  OR kran3Close.topStatus
  OR kran5Open.topStatus
  OR error_Krans.topStatus
  OR pnsOn.topStatus
  OR Pg_VhodLessThen300.topStatus
  OR Pg_VyhodLessThen300.topStatus
  OR nu1Off.topStatus
  OR nu2Off.topStatus
  OR autoNuOff.topStatus
  OR timer600.topStatus
  OR Avom1Off.topStatus
  OR Avom2Off.topStatus
  OR Avom3Off.topStatus
  OR Avom4Off.topStatus
  OR autoAVOMOff.topStatus
  OR timer5.topStatus
  OR runUnsuccessful.topStatus;
  (*OR klapan1.topStatus
  OR klapan2.topStatus;*)

  (*TODO: TYPE PROGRAM CODE HERE*)
  StrAlg.status :=  SHL(BYTE_TO_DWORD(source_for_Status), 29)
  			OR SHL(BYTE_TO_DWORD(cmd_for_Status), 26)
  			OR SHL(BYTE_TO_DWORD(command_error_for_Status), 23)
  			OR SHL(BOOL_TO_DWORD(StrAlg.OpcCommandsDisabled ), 21)
  			OR SHL(BOOL_TO_DWORD(StrAlg.hasError),4)
  			OR SHL(BOOL_TO_DWORD(StrAlg.CanRun),2)
  			OR SHL(BOOL_TO_DWORD(StrAlg.isEnded),1)
  			OR BOOL_TO_DWORD(StrAlg.isRuning);
END_FUNCTION_BLOCK

FUNCTION_BLOCK ppuAlg
  VAR_IN_OUT
    StrAlg : struct_Alg;
    StrPermis : ppu_permissions;
  END_VAR
  VAR
    Level_masla_Norm : struct_PhaseAlgoritm;
    T_masla_Norm : struct_PhaseAlgoritm;
    Krans_ready_to_move : struct_PhaseAlgoritm;
    Krans_Poloj : struct_PhaseAlgoritm;
    Net_AO_KC_SHKS04M : struct_PhaseAlgoritm;
    EGPA_Stop : struct_PhaseAlgoritm;
    Naprajenie_ZRU : struct_PhaseAlgoritm;
    All_IM_Off : struct_PhaseAlgoritm;
    Nalichie_PitanieSHU : struct_PhaseAlgoritm;
    CU_IM_Norm : struct_PhaseAlgoritm;
    MV_Poloj_RolledON : struct_PhaseAlgoritm;
    MV_Poloj_RolledOFF : struct_PhaseAlgoritm;
    NOTAnalogNS : struct_PhaseAlgoritm;
    Net_ASPS_Analogs : struct_PhaseAlgoritm;
    Remont_Not : struct_PhaseAlgoritm;
    not_AS : struct_PhaseAlgoritm;
    Gotov_Vozb : struct_PhaseAlgoritm;
    dP_kr1 : struct_PhaseAlgoritm;
    Auto_Rej : struct_PhaseAlgoritm;
    CK_IM_norm : struct_PhaseAlgoritm;
    Impuls_Gaz : struct_PhaseAlgoritm;
    Est_rezerv_NU : struct_PhaseAlgoritm;
    fb_Level_masla_Norm : fb_ph_CustomPhase;
    fb_T_masla_Norm : fb_ph_CustomPhase;
    fb_Krans_ready_to_move : fb_ph_CustomPhase;
    fb_Not_AS_PS : fb_ph_CustomPhase;
    fb_Not_AO_NO_EAO : fb_ph_CustomPhase;
    fb_Krans_Poloj : fb_ph_CustomPhase;
    fb_Net_AO_KC_SHKS04M : fb_ph_CustomPhase;
    fb_EGPA_Stop : fb_ph_CustomPhase;
    fb_Naprajenie_ZRU : fb_ph_CustomPhase;
    fb_All_IM_Off : fb_ph_CustomPhase;
    fb_Nalichie_PitanieSHU : fb_ph_CustomPhase;
    fb_CU_IM_Norm : fb_ph_CustomPhase;
    fb_MV_Poloj_RolledON : fb_ph_CustomPhase;
    fb_MV_Poloj_RolledOFF : fb_ph_CustomPhase;
    fb_NOTAnalogNS : fb_ph_CustomPhase;
    fb_Net_ASPS_Analogs : fb_ph_CustomPhase;
    fb_Remont_Not : fb_ph_CustomPhase;
    fb_not_AS : fb_ph_CustomPhase;
    fb_Gotov_Vozb : fb_ph_CustomPhase;
    fb_dP_kr1 : fb_ph_CustomPhase;
    fb_Auto_Rej : fb_ph_CustomPhase;
    fb_CK_IM_norm : fb_ph_CustomPhase;
    fb_Impuls_Gaz : fb_ph_CustomPhase;
    fb_Est_rezerv_NU : fb_ph_CustomPhase;
    _sunpackerCommand : fb_sunpackerCommand;
    _statusAi : TYPE_StatusAi;
    _statusDualInput : TYPE_statusDualInput;
    _DualStateImAction : TYPE_DualStateImAction;
    _PhaseAlgoritmAction : TYPE_PhaseAlgoritmAction;
    _basketStats : TYPE_basketStats;
    source : BYTE;
    cmd : BYTE;
    lastCmd : BYTE;
    source_for_Status : BYTE;
    cmd_for_Status : BYTE;
    command_error_for_Status : BYTE;
    resetCmdTimer : TON;
    resetCmdTimerPriznak : BOOL;
    onInit : BOOL;
  END_VAR
  VAR_EXTERNAL
    IM : ImConfig;
    ai : AiConfig;
    di : DiConfig;
    algManager : struct_AlgoritmsManager;
    protectManager : struct_ProtectionsManager;
    NotHasRezervNU : BOOL;
    algoritms : AlgoritmsConfig;
    modegpa : TYPE_ModeGpa;
  END_VAR

  IF NOT onInit THEN
            fb_Level_masla_Norm(phaseNumber:=0);
                fb_T_masla_Norm(phaseNumber:=1);
         fb_Krans_ready_to_move(phaseNumber:=2);
                 fb_Krans_Poloj(phaseNumber:=3);
           fb_Net_AO_KC_SHKS04M(phaseNumber:=4);
                   fb_EGPA_Stop(phaseNumber:=5);
              fb_Naprajenie_ZRU(phaseNumber:=6);
                  fb_All_IM_Off(phaseNumber:=7);
         fb_Nalichie_PitanieSHU(phaseNumber:=8);
                  fb_CU_IM_Norm(phaseNumber:=9);
           fb_MV_Poloj_RolledON(phaseNumber:=10);
          fb_MV_Poloj_RolledOFF(phaseNumber:=11);
                 fb_NOTAnalogNS(phaseNumber:=12);
            fb_Net_ASPS_Analogs(phaseNumber:=13);
                  fb_Remont_Not(phaseNumber:=14);
                      fb_not_AS(phaseNumber:=15);
                  fb_Gotov_Vozb(phaseNumber:=16);
                      fb_dP_kr1(phaseNumber:=17);
                    fb_Auto_Rej(phaseNumber:=18);
                  fb_CK_IM_norm(phaseNumber:=19);
                  fb_Impuls_Gaz(phaseNumber:=20);
               fb_Est_rezerv_NU(phaseNumber:=21);

  onInit:=TRUE;
  END_IF;

            fb_Level_masla_Norm(StrPh:=Level_masla_Norm);
                fb_T_masla_Norm(StrPh:=T_masla_Norm);
         fb_Krans_ready_to_move(StrPh:=Krans_ready_to_move);
                 fb_Krans_Poloj(StrPh:=Krans_Poloj);
           fb_Net_AO_KC_SHKS04M(StrPh:=Net_AO_KC_SHKS04M);
                   fb_EGPA_Stop(StrPh:=EGPA_Stop);
              fb_Naprajenie_ZRU(StrPh:=Naprajenie_ZRU);
                  fb_All_IM_Off(StrPh:=All_IM_Off);
         fb_Nalichie_PitanieSHU(StrPh:=Nalichie_PitanieSHU);
                  fb_CU_IM_Norm(StrPh:=CU_IM_Norm);
           fb_MV_Poloj_RolledON(StrPh:=MV_Poloj_RolledON);
          fb_MV_Poloj_RolledOFF(StrPh:=MV_Poloj_RolledOFF);
                 fb_NOTAnalogNS(StrPh:=NOTAnalogNS);
            fb_Net_ASPS_Analogs(StrPh:=Net_ASPS_Analogs);
                  fb_Remont_Not(StrPh:=Remont_Not);
                      fb_not_AS(StrPh:=not_AS);
                  fb_Gotov_Vozb(StrPh:=Gotov_Vozb);
                      fb_dP_kr1(StrPh:=dP_kr1);
                    fb_Auto_Rej(StrPh:=Auto_Rej);
                  fb_CK_IM_norm(StrPh:=CK_IM_norm);
                  fb_Impuls_Gaz(StrPh:=Impuls_Gaz);
               fb_Est_rezerv_NU(StrPh:=Est_rezerv_NU);

  IF StrAlg.isRuning THEN

  (*Нет неисправных аналогов*)
  NOTAnalogNS.top:= NOT analogsNS();

  (*уровень масла в норме*)
  Level_masla_Norm.top:= (ai.Yroven_masla_v_maslobake.interval = _statusAi.normal);

  (*температура масла в норме*)
  T_masla_Norm.top:=(ai.T_masla_v_maslobake.interval=_statusAi.normal);

  (*Краны готовы к управлению*)
  Krans_ready_to_move.top:= 	NOT (im.kran1.so OR im.kran1.sz OR
                                     im.kran2.so OR im.kran2.sz OR
                                     im.kran3.so OR im.kran3.sz OR
                                     im.kran3b.so OR im.kran3b.sz OR
                                     im.kran4.so OR im.kran4.sz OR
  			     im.kran5.so OR im.kran5.sz OR
                                     im.kran6.so OR im.kran6.sz);

  (* Режим ЭГПА остановлен *)
  EGPA_Stop.top:=	(algmanager.mode = modegpa.MODE_STOP);

  (*Нет АС ПС по Аналогам*)
  Net_ASPS_Analogs.top:= NOT (algManager.analogsPS OR algManager.ProtectionSignaling);

  (*Есть напряжение в ЗРУ*)
  Nalichie_PitanieSHU.top:=	im.SingleSignals.Neisprav_BP_1.Q AND
                                im.singleSignals.Neisprav_BP_2.Q AND
                                im.singleSignals.Neisprav_BP_3.Q AND
                                im.singleSignals.Neisprav_BP_4.Q AND
                                im.singleSignals.Neisprav_BP_5.Q AND
                                im.singleSignals.Neisprav_BP_6.Q AND
                                im.singleSignals.Neisprav_BP_7.Q AND
  			im.singleSignals.Neisprav_BP_8.Q AND
                                im.singleSignals.Neisprav_BP_9.Q AND
                                im.singleSignals.Neisprav_BP_10.Q AND
                                im.singleSignals.Nalichie_220_perem_vhod_v_SHY.Q AND
                                im.singleSignals.Nalichie_220_post_vhod_v_SHY.Q AND
  			im.singleSignals.BEAO_vkl.Q;

  (*Есть напряжение в ЗРУ*)
  Naprajenie_ZRU.top:= im.singleSignals.Nalichie_220_post_na_shinah_ypr_ZRY.Q;

  (*Наличие ЦУ ИМ*)
  CU_IM_Norm.top:= NOT nsCepeiUpravlenya(im);

  (*ИМ отключены*)
  All_IM_Off.top:=(im.MB.onStatus=_statusDualInput.STATUS_OFF) AND
                  (im.pns.onStatus=_statusDualInput.STATUS_OFF) AND
                  (im.nu1.onStatus=_statusDualInput.STATUS_OFF) AND
  	      (im.nu2.onStatus=_statusDualInput.STATUS_OFF) AND
                  (im.v1_Avom.onStatus=_statusDualInput.STATUS_OFF) AND
                  (im.v2_Avom.onStatus=_statusDualInput.STATUS_OFF) AND
                  (im.v3_Avom.onStatus=_statusDualInput.STATUS_OFF) AND
                  (im.v4_Avom.onStatus=_statusDualInput.STATUS_OFF) AND
                  (im.CMN_pump.onStatus=_statusDualInput.STATUS_OFF) AND
  	      (im.Ten_MB.onStatus=_statusDualInput.STATUS_OFF) AND
                  (im.Ten_kollect.onStatus=_statusDualInput.STATUS_OFF) AND
                  (im.Kalorifer_ABO.onStatus=_statusDualInput.STATUS_OFF);

  (*Нет АО от ШКС*)
  Net_AO_KC_SHKS04M.top:= NOT Im.singleSignals.AO_KC_ot_SHKC_04M.Q AND Im.singleSignals.AO_KC_ot_SHKC_04M.reliability;

  (*Наличие автоматического режима насосов*)
  Auto_Rej.top:= im.nu1.Auto AND im.nu2.Auto AND im.pns.Auto;

  Krans_Poloj.top:=		(Im.kran1.onStatus=_statusDualInput.STATUS_OFF) AND
  			(Im.kran2.onStatus=_statusDualInput.STATUS_OFF) AND
  			(Im.kran3.onStatus=_statusDualInput.STATUS_OFF) AND
  			(Im.kran3b.onStatus=_statusDualInput.STATUS_ON) AND
  			(Im.kran4.onStatus=_statusDualInput.STATUS_OFF) AND
  			(Im.kran5.onStatus=_statusDualInput.STATUS_ON) AND
  			(Im.kran6.onStatus=_statusDualInput.STATUS_ON);

  (*Тележка МВ вкачена*)
  MV_Poloj_RolledON.top:= im.MB.basketStatus = _basketStats.BASKET_ROLLEDIN;

  (*Тележка МВ выкачена*)
  MV_Poloj_RolledOFF.top:= im.MB.basketStatus = _basketStats.BASKET_ROLLEDOUT;

  (*Готовность возбудителя*)
  Gotov_Vozb.top:= im.singleSignals.Gotovnosst_vozb.Q;

  (*Нет сигнала перепада на кране 1*)
  dP_kr1.top:= ((im.singleSignals.dP_gaza_kr_1.Q) AND (im.singleSignals.dP_gaza_kr_1.reliability));

  (*Давление импульсного газа в норме*)
  Impuls_Gaz.top:=(ai.Davlenie_impylsnogo_gaza.interval=_statusAi.normal);

  (*Нет защит в ремонте*)
  Remont_Not.top:=not protectManager.protectionInRemont;

  CK_IM_norm.top:= not nsCepeiControl(IM);

  not_AS.top:=NOT (algManager.DiscretPS OR algManager.analogsPS OR algManager.ProtectionSignaling);

  Est_rezerv_NU.top:= NOT NotHasRezervNU;

  (*ППУ для первого этапа пуска*)
  StrPermis.ppuFirst_for_Pusk:= NOTAnalogNS.top AND
  			Level_masla_Norm.top AND
  			T_masla_Norm.top AND
  			Krans_ready_to_move.top AND
  			EGPA_Stop.top AND
  			Net_ASPS_Analogs.top AND
  			Nalichie_PitanieSHU.top AND
  			Naprajenie_ZRU.top AND
  			CU_IM_Norm.top AND
  			All_IM_Off.top AND
  			Net_AO_KC_SHKS04M.top AND
  			Auto_Rej.top AND
  			Krans_Poloj.top AND
  			MV_Poloj_RolledON.top AND
  			Gotov_Vozb.top AND
  			dP_kr1.top AND
  			Impuls_Gaz.top AND
                                Remont_Not.top AND
                                CK_IM_norm.top AND
                                not_AS.top;

  (*ППУ для проверки двигателя*)
  StrPermis.ppuFirst_for_V:=
  			NOTAnalogNS.top AND
  			Level_masla_Norm.top AND
  			T_masla_Norm.top AND
  			EGPA_Stop.top AND
  			Net_ASPS_Analogs.top AND
  			Nalichie_PitanieSHU.top AND
  			Naprajenie_ZRU.top AND
  			CU_IM_Norm.top AND
  			All_IM_Off.top AND
  			Net_AO_KC_SHKS04M.top AND
  			Auto_Rej.top AND
  			MV_Poloj_RolledON.top AND
  			Gotov_Vozb.top AND
                                Remont_Not.top AND
                                CK_IM_norm.top AND
                                not_AS.top;

  (*ППУ для проверки масла смазки и масло газ*)
  StrPermis.ppuFirst_for_Pms_dPmg:=
  			NOTAnalogNS.top AND
  			Level_masla_Norm.top AND
  			T_masla_Norm.top AND
  			EGPA_Stop.top AND
  			Net_ASPS_Analogs.top AND
  			Nalichie_PitanieSHU.top AND
  			CU_IM_Norm.top AND
  			All_IM_Off.top AND
  			Net_AO_KC_SHKS04M.top AND
  			Auto_Rej.top AND
  			MV_Poloj_RolledOFF.top AND
                                Remont_Not.top AND
                                CK_IM_norm.top AND
                                not_AS.top;

  (*ППУ проверки кранов*)
  StrPermis.ppuFirst_for_K:=
  			NOTAnalogNS.top AND
  			Level_masla_Norm.top AND
  			T_masla_Norm.top AND
  			Krans_ready_to_move.top AND
  			EGPA_Stop.top AND
  			Net_ASPS_Analogs.top AND
  			Nalichie_PitanieSHU.top AND
  			Naprajenie_ZRU.top AND
  			CU_IM_Norm.top AND
  			All_IM_Off.top AND
  			Net_AO_KC_SHKS04M.top AND
  			Auto_Rej.top AND
  			Krans_Poloj.top AND
  			MV_Poloj_RolledOFF.top AND
  			dP_kr1.top AND
  			Impuls_Gaz.top AND
                                Remont_Not.top AND
                                CK_IM_norm.top AND
                                not_AS.top;

  (*ППУ имитация пуска*)
  StrPermis.ppuFirst_for_I:=
  			NOTAnalogNS.top AND
  			Level_masla_Norm.top AND
  			T_masla_Norm.top AND
  			Krans_ready_to_move.top AND
  			EGPA_Stop.top AND
  			Net_ASPS_Analogs.top AND
  			Nalichie_PitanieSHU.top AND
  			Naprajenie_ZRU.top AND
  			CU_IM_Norm.top AND
  			All_IM_Off.top AND
  			Net_AO_KC_SHKS04M.top AND
  			Auto_Rej.top AND
  			Krans_Poloj.top AND
  			MV_Poloj_RolledOn.top AND
  			dP_kr1.top AND
  			Impuls_Gaz.top AND
                                Gotov_Vozb.top AND
                                Remont_Not.top AND
                                CK_IM_norm.top AND
                                not_AS.top;

  (*ППУ для второго этапа пуска в режиме "ПУск" и "Режим В"*)
  StrPermis.ppuSecond_V_Pusk:=

  			Level_masla_Norm.top AND
  			T_masla_Norm.top AND
  			Nalichie_PitanieSHU.top AND
  			Naprajenie_ZRU.top AND
  			Net_AO_KC_SHKS04M.top AND
  			Auto_Rej.top AND
  			MV_Poloj_RolledON.top AND
  			Gotov_Vozb.top AND
                                Remont_Not.top AND
                                CK_IM_norm.top AND not_AS.top
                                AND (algmanager.mode=modegpa.MODE_APUSK)
                                 OR (algmanager.mode=modegpa.MODE_MPUSK)
                                 OR (algmanager.mode=modegpa.MODE_PUSKV);
